   DATA[2032,33] := 0.3084905;
   DATA[2032,34] := 2.0;
   DATA[2032,35] := 250.2243;
   DATA[2032,36] := 1.69801;
   DATA[2032,37] := 189.1022;
   DATA[2032,38] := 0.000128152;
   DATA[2032,39] := 1.0;
   DATA[2032,40] := 1.0;
   DATA[2033,0] := 2.493034;
   DATA[2033,1] := 862.4616;
   DATA[2033,2] := 2.0;
   DATA[2033,3] := 2.0;
   DATA[2033,4] := 262.3686;
   DATA[2033,5] := 8.395155;
   DATA[2033,6] := 331.1971;
   DATA[2033,7] := 2.462179;
   DATA[2033,8] := 2.0;
   DATA[2033,9] := 2.0;
   DATA[2033,10] := 2.0;
   DATA[2033,11] := 19.76759;
   DATA[2033,12] := 2.209653;
   DATA[2033,13] := 801.3971;
   DATA[2033,14] := 1.0;
   DATA[2033,15] := 2.0;
   DATA[2033,16] := 1.0;
   DATA[2033,17] := 1.0;
   DATA[2033,18] := 1.0;
   DATA[2033,19] := 2.0;
   DATA[2033,20] := 148.808;
   DATA[2033,21] := 154.8834;
   DATA[2033,22] := 1.717361;
   DATA[2033,23] := 830.7485;
   DATA[2033,24] := 2.0;
   DATA[2033,25] := 2.0;
   DATA[2033,26] := 7.874455;
   DATA[2033,27] := 143.9375;
   DATA[2033,28] := 262.1764;
   DATA[2033,29] := 12.07383;
   DATA[2033,30] := 1.726609;
   DATA[2033,31] := 1.281798;
   DATA[2033,32] := 0.7355248;
   DATA[2033,33] := 0.3084905;
   DATA[2033,34] := 2.0;
   DATA[2033,35] := 250.2243;
   DATA[2033,36] := 1.69801;
   DATA[2033,37] := 189.0381;
   DATA[2033,38] := 0.000128152;
   DATA[2033,39] := 1.0;
   DATA[2033,40] := 1.0;
   DATA[2034,0] := 2.47702;
   DATA[2034,1] := 862.2653;
   DATA[2034,2] := 2.0;
   DATA[2034,3] := 2.0;
   DATA[2034,4] := 262.3686;
   DATA[2034,5] := 8.395155;
   DATA[2034,6] := 331.1971;
   DATA[2034,7] := 2.46282;
   DATA[2034,8] := 2.0;
   DATA[2034,9] := 2.0;
   DATA[2034,10] := 2.0;
   DATA[2034,11] := 19.74198;
   DATA[2034,12] := 2.208756;
   DATA[2034,13] := 801.6775;
   DATA[2034,14] := 1.0;
   DATA[2034,15] := 2.0;
   DATA[2034,16] := 1.0;
   DATA[2034,17] := 1.0;
   DATA[2034,18] := 1.0;
   DATA[2034,19] := 2.0;
   DATA[2034,20] := 148.808;
   DATA[2034,21] := 154.6783;
   DATA[2034,22] := 1.717361;
   DATA[2034,23] := 830.5947;
   DATA[2034,24] := 2.0;
   DATA[2034,25] := 2.0;
   DATA[2034,26] := 7.874455;
   DATA[2034,27] := 143.9375;
   DATA[2034,28] := 261.888;
   DATA[2034,29] := 12.07383;
   DATA[2034,30] := 1.725327;
   DATA[2034,31] := 1.277699;
   DATA[2034,32] := 0.7355248;
   DATA[2034,33] := 0.3084905;
   DATA[2034,34] := 2.0;
   DATA[2034,35] := 250.0641;
   DATA[2034,36] := 1.69801;
   DATA[2034,37] := 188.8779;
   DATA[2034,38] := 0.000128152;
   DATA[2034,39] := 1.0;
   DATA[2034,40] := 1.0;
   DATA[2035,0] := 2.456202;
   DATA[2035,1] := 862.1083;
   DATA[2035,2] := 2.0;
   DATA[2035,3] := 2.0;
   DATA[2035,4] := 262.3686;
   DATA[2035,5] := 8.395155;
   DATA[2035,6] := 331.1971;
   DATA[2035,7] := 2.46282;
   DATA[2035,8] := 2.0;
   DATA[2035,9] := 2.0;
   DATA[2035,10] := 2.0;
   DATA[2035,11] := 19.70997;
   DATA[2035,12] := 2.208756;
   DATA[2035,13] := 801.317;
   DATA[2035,14] := 1.0;
   DATA[2035,15] := 2.0;
   DATA[2035,16] := 1.0;
   DATA[2035,17] := 1.0;
   DATA[2035,18] := 1.0;
   DATA[2035,19] := 2.0;
   DATA[2035,20] := 148.808;
   DATA[2035,21] := 154.6783;
   DATA[2035,22] := 1.717361;
   DATA[2035,23] := 830.5563;
   DATA[2035,24] := 2.0;
   DATA[2035,25] := 2.0;
   DATA[2035,26] := 7.874455;
   DATA[2035,27] := 143.9375;
   DATA[2035,28] := 261.888;
   DATA[2035,29] := 12.07383;
   DATA[2035,30] := 1.723532;
   DATA[2035,31] := 1.260535;
   DATA[2035,32] := 0.7355248;
   DATA[2035,33] := 0.3084905;
   DATA[2035,34] := 2.0;
   DATA[2035,35] := 249.8558;
   DATA[2035,36] := 1.69801;
   DATA[2035,37] := 188.8138;
   DATA[2035,38] := 0.000128152;
   DATA[2035,39] := 1.0;
   DATA[2035,40] := 1.0;
   DATA[2036,0] := 2.445953;
   DATA[2036,1] := 862.2653;
   DATA[2036,2] := 2.0;
   DATA[2036,3] := 2.0;
   DATA[2036,4] := 262.3686;
   DATA[2036,5] := 8.395155;
   DATA[2036,6] := 331.1971;
   DATA[2036,7] := 2.463204;
   DATA[2036,8] := 2.0;
   DATA[2036,9] := 2.0;
   DATA[2036,10] := 2.0;
   DATA[2036,11] := 19.70997;
   DATA[2036,12] := 2.208756;
   DATA[2036,13] := 801.0767;
   DATA[2036,14] := 1.0;
   DATA[2036,15] := 2.0;
   DATA[2036,16] := 1.0;
   DATA[2036,17] := 1.0;
   DATA[2036,18] := 1.0;
   DATA[2036,19] := 2.0;
   DATA[2036,20] := 148.808;
   DATA[2036,21] := 154.6783;
   DATA[2036,22] := 1.716464;
   DATA[2036,23] := 831.1331;
   DATA[2036,24] := 2.0;
   DATA[2036,25] := 2.0;
   DATA[2036,26] := 7.874455;
   DATA[2036,27] := 143.9375;
   DATA[2036,28] := 261.888;
   DATA[2036,29] := 12.07383;
   DATA[2036,30] := 1.723532;
   DATA[2036,31] := 1.254259;
   DATA[2036,32] := 0.7355248;
   DATA[2036,33] := 0.3084905;
   DATA[2036,34] := 2.0;
   DATA[2036,35] := 249.8558;
   DATA[2036,36] := 1.69801;
   DATA[2036,37] := 188.8138;
   DATA[2036,38] := 0.000128152;
   DATA[2036,39] := 1.0;
   DATA[2036,40] := 1.0;
   DATA[2037,0] := 2.432822;
   DATA[2037,1] := 862.0691;
   DATA[2037,2] := 2.0;
   DATA[2037,3] := 2.0;
   DATA[2037,4] := 262.3686;
   DATA[2037,5] := 8.395155;
   DATA[2037,6] := 331.1971;
   DATA[2037,7] := 2.463589;
   DATA[2037,8] := 2.0;
   DATA[2037,9] := 2.0;
   DATA[2037,10] := 2.0;
   DATA[2037,11] := 19.75159;
   DATA[2037,12] := 2.208756;
   DATA[2037,13] := 801.1167;
   DATA[2037,14] := 1.0;
   DATA[2037,15] := 2.0;
   DATA[2037,16] := 1.0;
   DATA[2037,17] := 1.0;
   DATA[2037,18] := 1.0;
   DATA[2037,19] := 2.0;
   DATA[2037,20] := 148.808;
   DATA[2037,21] := 154.6783;
   DATA[2037,22] := 1.715824;
   DATA[2037,23] := 831.3253;
   DATA[2037,24] := 2.0;
   DATA[2037,25] := 2.0;
   DATA[2037,26] := 7.874455;
   DATA[2037,27] := 143.9375;
   DATA[2037,28] := 261.888;
   DATA[2037,29] := 12.07383;
   DATA[2037,30] := 1.723532;
   DATA[2037,31] := 1.241962;
   DATA[2037,32] := 0.7355248;
   DATA[2037,33] := 0.3077219;
   DATA[2037,34] := 2.0;
   DATA[2037,35] := 249.8558;
   DATA[2037,36] := 1.649953;
   DATA[2037,37] := 188.8138;
   DATA[2037,38] := 0.000128152;
   DATA[2037,39] := 1.0;
   DATA[2037,40] := 1.0;
   DATA[2038,0] := 2.432822;
   DATA[2038,1] := 862.0691;
   DATA[2038,2] := 2.0;
   DATA[2038,3] := 2.0;
   DATA[2038,4] := 262.3686;
   DATA[2038,5] := 8.395155;
   DATA[2038,6] := 331.1971;
   DATA[2038,7] := 2.463589;
   DATA[2038,8] := 2.0;
   DATA[2038,9] := 2.0;
   DATA[2038,10] := 2.0;
   DATA[2038,11] := 19.75159;
   DATA[2038,12] := 2.208756;
   DATA[2038,13] := 801.1167;
   DATA[2038,14] := 1.0;
   DATA[2038,15] := 2.0;
   DATA[2038,16] := 1.0;
   DATA[2038,17] := 1.0;
   DATA[2038,18] := 1.0;
   DATA[2038,19] := 2.0;
   DATA[2038,20] := 148.808;
   DATA[2038,21] := 154.6783;
   DATA[2038,22] := 1.715824;
   DATA[2038,23] := 831.3253;
   DATA[2038,24] := 2.0;
   DATA[2038,25] := 2.0;
   DATA[2038,26] := 7.874455;
   DATA[2038,27] := 143.9375;
   DATA[2038,28] := 261.888;
   DATA[2038,29] := 12.07383;
   DATA[2038,30] := 1.723532;
   DATA[2038,31] := 1.241962;
   DATA[2038,32] := 0.7355248;
   DATA[2038,33] := 0.3077219;
   DATA[2038,34] := 2.0;
   DATA[2038,35] := 249.8558;
   DATA[2038,36] := 1.649953;
   DATA[2038,37] := 188.8138;
   DATA[2038,38] := 0.000128152;
   DATA[2038,39] := 1.0;
   DATA[2038,40] := 1.0;
   DATA[2039,0] := 2.423213;
   DATA[2039,1] := 861.7158;
   DATA[2039,2] := 2.0;
   DATA[2039,3] := 2.0;
   DATA[2039,4] := 262.3686;
   DATA[2039,5] := 8.393232;
   DATA[2039,6] := 331.1971;
   DATA[2039,7] := 2.463589;
   DATA[2039,8] := 2.0;
   DATA[2039,9] := 2.0;
   DATA[2039,10] := 2.0;
   DATA[2039,11] := 19.77399;
   DATA[2039,12] := 2.210037;
   DATA[2039,13] := 800.9565;
   DATA[2039,14] := 1.0;
   DATA[2039,15] := 2.0;
   DATA[2039,16] := 1.0;
   DATA[2039,17] := 1.0;
   DATA[2039,18] := 1.0;
   DATA[2039,19] := 2.0;
   DATA[2039,20] := 148.808;
   DATA[2039,21] := 154.909;
   DATA[2039,22] := 1.715824;
   DATA[2039,23] := 831.3253;
   DATA[2039,24] := 2.0;
   DATA[2039,25] := 2.0;
   DATA[2039,26] := 7.874455;
   DATA[2039,27] := 143.9375;
   DATA[2039,28] := 261.888;
   DATA[2039,29] := 12.07383;
   DATA[2039,30] := 1.725455;
   DATA[2039,31] := 1.237351;
   DATA[2039,32] := 0.7355248;
   DATA[2039,33] := 0.3077219;
   DATA[2039,34] := 2.0;
   DATA[2039,35] := 250.032;
   DATA[2039,36] := 1.649953;
   DATA[2039,37] := 188.8138;
   DATA[2039,38] := 0.000128152;
   DATA[2039,39] := 1.0;
   DATA[2039,40] := 1.0;
   DATA[2040,0] := 2.423213;
   DATA[2040,1] := 862.0691;
   DATA[2040,2] := 2.0;
   DATA[2040,3] := 2.0;
   DATA[2040,4] := 262.3686;
   DATA[2040,5] := 8.393232;
   DATA[2040,6] := 331.1971;
   DATA[2040,7] := 2.463589;
   DATA[2040,8] := 2.0;
   DATA[2040,9] := 2.0;
   DATA[2040,10] := 2.0;
   DATA[2040,11] := 19.77399;
   DATA[2040,12] := 2.210037;
   DATA[2040,13] := 800.7562;
   DATA[2040,14] := 1.0;
   DATA[2040,15] := 2.0;
   DATA[2040,16] := 1.0;
   DATA[2040,17] := 1.0;
   DATA[2040,18] := 1.0;
   DATA[2040,19] := 2.0;
   DATA[2040,20] := 148.808;
   DATA[2040,21] := 155.0372;
   DATA[2040,22] := 1.715824;
   DATA[2040,23] := 831.556;
   DATA[2040,24] := 2.0;
   DATA[2040,25] := 2.0;
   DATA[2040,26] := 7.874455;
   DATA[2040,27] := 143.9375;
   DATA[2040,28] := 262.1764;
   DATA[2040,29] := 12.07383;
   DATA[2040,30] := 1.725583;
   DATA[2040,31] := 1.251953;
   DATA[2040,32] := 0.7355248;
   DATA[2040,33] := 0.3084905;
   DATA[2040,34] := 2.0;
   DATA[2040,35] := 250.0961;
   DATA[2040,36] := 1.649953;
   DATA[2040,37] := 188.9419;
   DATA[2040,38] := 0.000128152;
   DATA[2040,39] := 1.0;
   DATA[2040,40] := 1.0;
   DATA[2041,0] := 2.433783;
   DATA[2041,1] := 861.598;
   DATA[2041,2] := 2.0;
   DATA[2041,3] := 2.0;
   DATA[2041,4] := 262.3686;
   DATA[2041,5] := 8.393232;
   DATA[2041,6] := 331.0946;
   DATA[2041,7] := 2.463589;
   DATA[2041,8] := 2.0;
   DATA[2041,9] := 2.0;
   DATA[2041,10] := 2.0;
   DATA[2041,11] := 19.77399;
   DATA[2041,12] := 2.210037;
   DATA[2041,13] := 800.7162;
   DATA[2041,14] := 1.0;
   DATA[2041,15] := 2.0;
   DATA[2041,16] := 1.0;
   DATA[2041,17] := 1.0;
   DATA[2041,18] := 1.0;
   DATA[2041,19] := 2.0;
   DATA[2041,20] := 148.808;
   DATA[2041,21] := 155.0372;
   DATA[2041,22] := 1.718387;
   DATA[2041,23] := 831.5176;
   DATA[2041,24] := 2.0;
   DATA[2041,25] := 2.0;
   DATA[2041,26] := 7.874455;
   DATA[2041,27] := 143.9375;
   DATA[2041,28] := 262.1764;
   DATA[2041,29] := 12.07383;
   DATA[2041,30] := 1.726096;
   DATA[2041,31] := 1.267837;
   DATA[2041,32] := 0.7355248;
   DATA[2041,33] := 0.3084905;
   DATA[2041,34] := 2.0;
   DATA[2041,35] := 250.1923;
   DATA[2041,36] := 1.649953;
   DATA[2041,37] := 189.1342;
   DATA[2041,38] := 0.000128152;
   DATA[2041,39] := 1.0;
   DATA[2041,40] := 1.0;
   DATA[2042,0] := 2.487589;
   DATA[2042,1] := 861.6373;
   DATA[2042,2] := 2.0;
   DATA[2042,3] := 2.0;
   DATA[2042,4] := 262.3686;
   DATA[2042,5] := 8.393232;
   DATA[2042,6] := 331.0946;
   DATA[2042,7] := 2.463589;
   DATA[2042,8] := 2.0;
   DATA[2042,9] := 2.0;
   DATA[2042,10] := 2.0;
   DATA[2042,11] := 19.74198;
   DATA[2042,12] := 2.210037;
   DATA[2042,13] := 800.5159;
   DATA[2042,14] := 1.0;
   DATA[2042,15] := 2.0;
   DATA[2042,16] := 1.0;
   DATA[2042,17] := 1.0;
   DATA[2042,18] := 1.0;
   DATA[2042,19] := 2.0;
   DATA[2042,20] := 148.808;
   DATA[2042,21] := 154.8065;
   DATA[2042,22] := 1.718387;
   DATA[2042,23] := 831.7098;
   DATA[2042,24] := 2.0;
   DATA[2042,25] := 2.0;
   DATA[2042,26] := 7.874455;
   DATA[2042,27] := 143.9375;
   DATA[2042,28] := 262.1764;
   DATA[2042,29] := 12.07383;
   DATA[2042,30] := 1.728275;
   DATA[2042,31] := 1.280646;
   DATA[2042,32] := 0.7355248;
   DATA[2042,33] := 0.3070813;
   DATA[2042,34] := 2.0;
   DATA[2042,35] := 250.4005;
   DATA[2042,36] := 1.649953;
   DATA[2042,37] := 189.1662;
   DATA[2042,38] := 0.000128152;
   DATA[2042,39] := 1.0;
   DATA[2042,40] := 1.0;
   DATA[2043,0] := 2.531147;
   DATA[2043,1] := 861.3232;
   DATA[2043,2] := 2.0;
   DATA[2043,3] := 2.0;
   DATA[2043,4] := 262.3686;
   DATA[2043,5] := 8.393232;
   DATA[2043,6] := 331.0946;
   DATA[2043,7] := 2.461667;
   DATA[2043,8] := 2.0;
   DATA[2043,9] := 2.0;
   DATA[2043,10] := 2.0;
   DATA[2043,11] := 19.72598;
   DATA[2043,12] := 2.210037;
   DATA[2043,13] := 800.7162;
   DATA[2043,14] := 1.0;
   DATA[2043,15] := 2.0;
   DATA[2043,16] := 1.0;
   DATA[2043,17] := 1.0;
   DATA[2043,18] := 1.0;
   DATA[2043,19] := 2.0;
   DATA[2043,20] := 148.808;
   DATA[2043,21] := 154.8065;
   DATA[2043,22] := 1.718387;
   DATA[2043,23] := 831.556;
   DATA[2043,24] := 2.0;
   DATA[2043,25] := 2.0;
   DATA[2043,26] := 7.874455;
   DATA[2043,27] := 143.9375;
   DATA[2043,28] := 262.0802;
   DATA[2043,29] := 12.07383;
   DATA[2043,30] := 1.728275;
   DATA[2043,31] := 1.281798;
   DATA[2043,32] := 0.7355248;
   DATA[2043,33] := 0.3068251;
   DATA[2043,34] := 2.0;
   DATA[2043,35] := 250.4005;
   DATA[2043,36] := 1.649953;
   DATA[2043,37] := 189.1662;
   DATA[2043,38] := 0.000128152;
   DATA[2043,39] := 1.0;
   DATA[2043,40] := 1.0;
   DATA[2044,0] := 2.573744;
   DATA[2044,1] := 861.5195;
   DATA[2044,2] := 2.0;
   DATA[2044,3] := 2.0;
   DATA[2044,4] := 262.3686;
   DATA[2044,5] := 8.393232;
   DATA[2044,6] := 331.0946;
   DATA[2044,7] := 2.461667;
   DATA[2044,8] := 2.0;
   DATA[2044,9] := 2.0;
   DATA[2044,10] := 2.0;
   DATA[2044,11] := 19.72598;
   DATA[2044,12] := 2.210037;
   DATA[2044,13] := 800.5159;
   DATA[2044,14] := 1.0;
   DATA[2044,15] := 2.0;
   DATA[2044,16] := 1.0;
   DATA[2044,17] := 1.0;
   DATA[2044,18] := 1.0;
   DATA[2044,19] := 2.0;
   DATA[2044,20] := 148.808;
   DATA[2044,21] := 154.8065;
   DATA[2044,22] := 1.718387;
   DATA[2044,23] := 831.6329;
   DATA[2044,24] := 2.0;
   DATA[2044,25] := 2.0;
   DATA[2044,26] := 7.874455;
   DATA[2044,27] := 143.9375;
   DATA[2044,28] := 262.0802;
   DATA[2044,29] := 12.07383;
   DATA[2044,30] := 1.730069;
   DATA[2044,31] := 1.271935;
   DATA[2044,32] := 0.7355248;
   DATA[2044,33] := 0.3068251;
   DATA[2044,34] := 2.0;
   DATA[2044,35] := 250.4005;
   DATA[2044,36] := 1.746067;
   DATA[2044,37] := 189.2624;
   DATA[2044,38] := 0.000128152;
   DATA[2044,39] := 1.0;
   DATA[2044,40] := 1.0;
   DATA[2045,0] := 2.601928;
   DATA[2045,1] := 861.5195;
   DATA[2045,2] := 2.0;
   DATA[2045,3] := 2.0;
   DATA[2045,4] := 262.3686;
   DATA[2045,5] := 8.393232;
   DATA[2045,6] := 331.0946;
   DATA[2045,7] := 2.461667;
   DATA[2045,8] := 2.0;
   DATA[2045,9] := 2.0;
   DATA[2045,10] := 2.0;
   DATA[2045,11] := 19.72598;
   DATA[2045,12] := 2.210037;
   DATA[2045,13] := 800.3156;
   DATA[2045,14] := 1.0;
   DATA[2045,15] := 2.0;
   DATA[2045,16] := 1.0;
   DATA[2045,17] := 1.0;
   DATA[2045,18] := 1.0;
   DATA[2045,19] := 2.0;
   DATA[2045,20] := 148.808;
   DATA[2045,21] := 154.8065;
   DATA[2045,22] := 1.718387;
   DATA[2045,23] := 831.7867;
   DATA[2045,24] := 2.0;
   DATA[2045,25] := 2.0;
   DATA[2045,26] := 7.874455;
   DATA[2045,27] := 144.2451;
   DATA[2045,28] := 262.0802;
   DATA[2045,29] := 12.07383;
   DATA[2045,30] := 1.731351;
   DATA[2045,31] := 1.271935;
   DATA[2045,32] := 0.7355248;
   DATA[2045,33] := 0.3068251;
   DATA[2045,34] := 2.0;
   DATA[2045,35] := 250.5127;
   DATA[2045,36] := 1.762086;
   DATA[2045,37] := 189.2624;
   DATA[2045,38] := 0.000128152;
   DATA[2045,39] := 1.0;
   DATA[2045,40] := 1.0;
   DATA[2046,0] := 2.636198;
   DATA[2046,1] := 861.284;
   DATA[2046,2] := 2.0;
   DATA[2046,3] := 2.0;
   DATA[2046,4] := 262.3686;
   DATA[2046,5] := 8.393232;
   DATA[2046,6] := 331.0946;
   DATA[2046,7] := 2.461667;
   DATA[2046,8] := 2.0;
   DATA[2046,9] := 2.0;
   DATA[2046,10] := 2.0;
   DATA[2046,11] := 19.71957;
   DATA[2046,12] := 2.206963;
   DATA[2046,13] := 800.3958;
   DATA[2046,14] := 1.0;
   DATA[2046,15] := 2.0;
   DATA[2046,16] := 1.0;
   DATA[2046,17] := 1.0;
   DATA[2046,18] := 1.0;
   DATA[2046,19] := 2.0;
   DATA[2046,20] := 148.808;
   DATA[2046,21] := 154.8065;
   DATA[2046,22] := 1.718387;
   DATA[2046,23] := 832.3635;
   DATA[2046,24] := 2.0;
   DATA[2046,25] := 2.0;
   DATA[2046,26] := 7.874455;
   DATA[2046,27] := 144.2451;
   DATA[2046,28] := 262.0802;
   DATA[2046,29] := 12.07383;
   DATA[2046,30] := 1.731351;
   DATA[2046,31] := 1.271679;
   DATA[2046,32] := 0.7355248;
   DATA[2046,33] := 0.3068251;
   DATA[2046,34] := 2.0;
   DATA[2046,35] := 250.6409;
   DATA[2046,36] := 1.762086;
   DATA[2046,37] := 189.3585;
   DATA[2046,38] := 0.000128152;
   DATA[2046,39] := 1.0;
   DATA[2046,40] := 1.0;
   DATA[2047,0] := 2.653172;
   DATA[2047,1] := 861.441;
   DATA[2047,2] := 2.0;
   DATA[2047,3] := 2.0;
   DATA[2047,4] := 262.3686;
   DATA[2047,5] := 8.393232;
   DATA[2047,6] := 331.0946;
   DATA[2047,7] := 2.461667;
   DATA[2047,8] := 2.0;
   DATA[2047,9] := 2.0;
   DATA[2047,10] := 2.0;
   DATA[2047,11] := 19.71957;
   DATA[2047,12] := 2.206322;
   DATA[2047,13] := 800.3156;
   DATA[2047,14] := 1.0;
   DATA[2047,15] := 2.0;
   DATA[2047,16] := 1.0;
   DATA[2047,17] := 1.0;
   DATA[2047,18] := 1.0;
   DATA[2047,19] := 2.0;
   DATA[2047,20] := 148.808;
   DATA[2047,21] := 154.8065;
   DATA[2047,22] := 1.718387;
   DATA[2047,23] := 832.2866;
   DATA[2047,24] := 2.0;
   DATA[2047,25] := 2.0;
   DATA[2047,26] := 7.874455;
   DATA[2047,27] := 144.0913;
   DATA[2047,28] := 262.0802;
   DATA[2047,29] := 12.07383;
   DATA[2047,30] := 1.731351;
   DATA[2047,31] := 1.290637;
   DATA[2047,32] := 0.7355248;
   DATA[2047,33] := 0.3068251;
   DATA[2047,34] := 2.0;
   DATA[2047,35] := 250.6409;
   DATA[2047,36] := 1.681991;
   DATA[2047,37] := 189.4386;
   DATA[2047,38] := 0.000128152;
   DATA[2047,39] := 1.0;
   DATA[2047,40] := 1.0;
   DATA[2048,0] := 2.663421;
   DATA[2048,1] := 861.441;
   DATA[2048,2] := 2.0;
   DATA[2048,3] := 2.0;
   DATA[2048,4] := 262.3686;
   DATA[2048,5] := 8.393232;
   DATA[2048,6] := 331.0946;
   DATA[2048,7] := 2.461667;
   DATA[2048,8] := 2.0;
   DATA[2048,9] := 2.0;
   DATA[2048,10] := 2.0;
   DATA[2048,11] := 19.69396;
   DATA[2048,12] := 2.206322;
   DATA[2048,13] := 800.3156;
   DATA[2048,14] := 1.0;
   DATA[2048,15] := 2.0;
   DATA[2048,16] := 1.0;
   DATA[2048,17] := 1.0;
   DATA[2048,18] := 1.0;
   DATA[2048,19] := 2.0;
   DATA[2048,20] := 148.808;
   DATA[2048,21] := 155.0372;
   DATA[2048,22] := 1.718387;
   DATA[2048,23] := 832.3635;
   DATA[2048,24] := 2.0;
   DATA[2048,25] := 2.0;
   DATA[2048,26] := 7.874455;
   DATA[2048,27] := 143.8862;
   DATA[2048,28] := 262.0802;
   DATA[2048,29] := 12.07383;
   DATA[2048,30] := 1.731351;
   DATA[2048,31] := 1.291789;
   DATA[2048,32] := 0.7355248;
   DATA[2048,33] := 0.3063127;
   DATA[2048,34] := 2.0;
   DATA[2048,35] := 250.6248;
   DATA[2048,36] := 1.649953;
   DATA[2048,37] := 189.4386;
   DATA[2048,38] := 0.000128152;
   DATA[2048,39] := 1.0;
   DATA[2048,40] := 1.0;
   DATA[2049,0] := 2.664062;
   DATA[2049,1] := 861.284;
   DATA[2049,2] := 2.0;
   DATA[2049,3] := 2.0;
   DATA[2049,4] := 262.3686;
   DATA[2049,5] := 8.393232;
   DATA[2049,6] := 331.0946;
   DATA[2049,7] := 2.461667;
   DATA[2049,8] := 2.0;
   DATA[2049,9] := 2.0;
   DATA[2049,10] := 2.0;
   DATA[2049,11] := 19.67796;
   DATA[2049,12] := 2.206322;
   DATA[2049,13] := 800.596;
   DATA[2049,14] := 1.0;
   DATA[2049,15] := 2.0;
   DATA[2049,16] := 1.0;
   DATA[2049,17] := 1.0;
   DATA[2049,18] := 1.0;
   DATA[2049,19] := 2.0;
   DATA[2049,20] := 148.808;
   DATA[2049,21] := 155.0372;
   DATA[2049,22] := 1.715952;
   DATA[2049,23] := 832.9018;
   DATA[2049,24] := 2.0;
   DATA[2049,25] := 2.0;
   DATA[2049,26] := 7.874455;
   DATA[2049,27] := 143.8862;
   DATA[2049,28] := 262.0802;
   DATA[2049,29] := 12.07383;
   DATA[2049,30] := 1.730838;
   DATA[2049,31] := 1.291918;
   DATA[2049,32] := 0.7355248;
   DATA[2049,33] := 0.3063127;
   DATA[2049,34] := 2.0;
   DATA[2049,35] := 250.3525;
   DATA[2049,36] := 1.649953;
   DATA[2049,37] := 189.3265;
   DATA[2049,38] := 0.000128152;
   DATA[2049,39] := 1.0;
   DATA[2049,40] := 1.0;
   DATA[2050,0] := 2.628191;
   DATA[2050,1] := 861.6373;
   DATA[2050,2] := 2.0;
   DATA[2050,3] := 2.0;
   DATA[2050,4] := 262.3686;
   DATA[2050,5] := 8.393232;
   DATA[2050,6] := 331.0946;
   DATA[2050,7] := 2.463589;
   DATA[2050,8] := 2.0;
   DATA[2050,9] := 2.0;
   DATA[2050,10] := 2.0;
   DATA[2050,11] := 19.67796;
   DATA[2050,12] := 2.206322;
   DATA[2050,13] := 800.7162;
   DATA[2050,14] := 1.0;
   DATA[2050,15] := 2.0;
   DATA[2050,16] := 1.0;
   DATA[2050,17] := 1.0;
   DATA[2050,18] := 1.0;
   DATA[2050,19] := 2.0;
   DATA[2050,20] := 148.808;
   DATA[2050,21] := 155.0372;
   DATA[2050,22] := 1.715952;
   DATA[2050,23] := 832.7095;
   DATA[2050,24] := 2.0;
   DATA[2050,25] := 2.0;
   DATA[2050,26] := 7.874455;
   DATA[2050,27] := 143.8862;
   DATA[2050,28] := 262.0802;
   DATA[2050,29] := 12.07383;
   DATA[2050,30] := 1.728019;
   DATA[2050,31] := 1.286922;
   DATA[2050,32] := 0.7355248;
   DATA[2050,33] := 0.3063127;
   DATA[2050,34] := 2.0;
   DATA[2050,35] := 250.3525;
   DATA[2050,36] := 1.649953;
   DATA[2050,37] := 189.1823;
   DATA[2050,38] := 0.000128152;
   DATA[2050,39] := 1.0;
   DATA[2050,40] := 1.0;
   DATA[2051,0] := 2.620824;
   DATA[2051,1] := 861.441;
   DATA[2051,2] := 2.0;
   DATA[2051,3] := 2.0;
   DATA[2051,4] := 262.3686;
   DATA[2051,5] := 8.392271;
   DATA[2051,6] := 331.0946;
   DATA[2051,7] := 2.463589;
   DATA[2051,8] := 2.0;
   DATA[2051,9] := 2.0;
   DATA[2051,10] := 2.0;
   DATA[2051,11] := 19.67796;
   DATA[2051,12] := 2.206322;
   DATA[2051,13] := 800.7963;
   DATA[2051,14] := 1.0;
   DATA[2051,15] := 2.0;
   DATA[2051,16] := 1.0;
   DATA[2051,17] := 1.0;
   DATA[2051,18] := 1.0;
   DATA[2051,19] := 2.0;
   DATA[2051,20] := 148.808;
   DATA[2051,21] := 155.0372;
   DATA[2051,22] := 1.715952;
   DATA[2051,23] := 833.171;
   DATA[2051,24] := 2.0;
   DATA[2051,25] := 2.0;
   DATA[2051,26] := 7.874455;
   DATA[2051,27] := 143.8862;
   DATA[2051,28] := 262.0802;
   DATA[2051,29] := 12.07383;
   DATA[2051,30] := 1.726865;
   DATA[2051,31] := 1.280902;
   DATA[2051,32] := 0.7355248;
   DATA[2051,33] := 0.3063127;
   DATA[2051,34] := 2.0;
   DATA[2051,35] := 250.3525;
   DATA[2051,36] := 1.649953;
   DATA[2051,37] := 189.1022;
   DATA[2051,38] := 0.000128152;
   DATA[2051,39] := 1.0;
   DATA[2051,40] := 1.0;
   DATA[2052,0] := 2.61538;
   DATA[2052,1] := 861.6765;
   DATA[2052,2] := 2.0;
   DATA[2052,3] := 2.0;
   DATA[2052,4] := 262.3686;
   DATA[2052,5] := 8.392271;
   DATA[2052,6] := 331.0946;
   DATA[2052,7] := 2.465127;
   DATA[2052,8] := 2.0;
   DATA[2052,9] := 2.0;
   DATA[2052,10] := 2.0;
   DATA[2052,11] := 19.62674;
   DATA[2052,12] := 2.206707;
   DATA[2052,13] := 801.1167;
   DATA[2052,14] := 1.0;
   DATA[2052,15] := 2.0;
   DATA[2052,16] := 1.0;
   DATA[2052,17] := 1.0;
   DATA[2052,18] := 1.0;
   DATA[2052,19] := 2.0;
   DATA[2052,20] := 148.808;
   DATA[2052,21] := 155.0372;
   DATA[2052,22] := 1.715952;
   DATA[2052,23] := 832.9787;
   DATA[2052,24] := 2.0;
   DATA[2052,25] := 2.0;
   DATA[2052,26] := 7.874455;
   DATA[2052,27] := 143.9631;
   DATA[2052,28] := 262.0802;
   DATA[2052,29] := 12.07383;
   DATA[2052,30] := 1.726609;
   DATA[2052,31] := 1.280902;
   DATA[2052,32] := 0.7355248;
   DATA[2052,33] := 0.3084265;
   DATA[2052,34] := 2.0;
   DATA[2052,35] := 250.3044;
   DATA[2052,36] := 1.649953;
   DATA[2052,37] := 189.1022;
   DATA[2052,38] := 0.000128152;
   DATA[2052,39] := 1.0;
   DATA[2052,40] := 1.0;
   DATA[2053,0] := 2.606732;
   DATA[2053,1] := 861.284;
   DATA[2053,2] := 2.0;
   DATA[2053,3] := 2.0;
   DATA[2053,4] := 262.3686;
   DATA[2053,5] := 8.392271;
   DATA[2053,6] := 331.0946;
   DATA[2053,7] := 2.465127;
   DATA[2053,8] := 2.0;
   DATA[2053,9] := 2.0;
   DATA[2053,10] := 2.0;
   DATA[2053,11] := 19.62674;
   DATA[2053,12] := 2.207091;
   DATA[2053,13] := 800.7963;
   DATA[2053,14] := 1.0;
   DATA[2053,15] := 2.0;
   DATA[2053,16] := 1.0;
   DATA[2053,17] := 1.0;
   DATA[2053,18] := 1.0;
   DATA[2053,19] := 2.0;
   DATA[2053,20] := 148.808;
   DATA[2053,21] := 155.0372;
   DATA[2053,22] := 1.716592;
   DATA[2053,23] := 833.1325;
   DATA[2053,24] := 2.0;
   DATA[2053,25] := 2.0;
   DATA[2053,26] := 7.874455;
   DATA[2053,27] := 143.9631;
   DATA[2053,28] := 262.0802;
   DATA[2053,29] := 12.07383;
   DATA[2053,30] := 1.726609;
   DATA[2053,31] := 1.274881;
   DATA[2053,32] := 0.7355248;
   DATA[2053,33] := 0.3084265;
   DATA[2053,34] := 2.0;
   DATA[2053,35] := 250.3044;
   DATA[2053,36] := 1.730048;
   DATA[2053,37] := 189.1022;
   DATA[2053,38] := 0.000128152;
   DATA[2053,39] := 1.0;
   DATA[2053,40] := 1.0;
   DATA[2054,0] := 2.582071;
   DATA[2054,1] := 861.5195;
   DATA[2054,2] := 2.0;
   DATA[2054,3] := 2.0;
   DATA[2054,4] := 262.3686;
   DATA[2054,5] := 8.392271;
   DATA[2054,6] := 331.0946;
   DATA[2054,7] := 2.464742;
   DATA[2054,8] := 2.0;
   DATA[2054,9] := 2.0;
   DATA[2054,10] := 2.0;
   DATA[2054,11] := 19.62674;
   DATA[2054,12] := 2.209013;
   DATA[2054,13] := 801.3971;
   DATA[2054,14] := 1.0;
   DATA[2054,15] := 2.0;
   DATA[2054,16] := 1.0;
   DATA[2054,17] := 1.0;
   DATA[2054,18] := 1.0;
   DATA[2054,19] := 2.0;
   DATA[2054,20] := 148.808;
   DATA[2054,21] := 155.0372;
   DATA[2054,22] := 1.717361;
   DATA[2054,23] := 832.9402;
   DATA[2054,24] := 2.0;
   DATA[2054,25] := 2.0;
   DATA[2054,26] := 7.874455;
   DATA[2054,27] := 143.9631;
   DATA[2054,28] := 262.0802;
   DATA[2054,29] := 12.07383;
   DATA[2054,30] := 1.726609;
   DATA[2054,31] := 1.276162;
   DATA[2054,32] := 0.7355248;
   DATA[2054,33] := 0.3084265;
   DATA[2054,34] := 2.0;
   DATA[2054,35] := 250.3044;
   DATA[2054,36] := 1.730048;
   DATA[2054,37] := 189.1022;
   DATA[2054,38] := 0.000128152;
   DATA[2054,39] := 1.0;
   DATA[2054,40] := 1.0;
   DATA[2055,0] := 2.564456;
   DATA[2055,1] := 861.284;
   DATA[2055,2] := 2.0;
   DATA[2055,3] := 2.0;
   DATA[2055,4] := 262.3686;
   DATA[2055,5] := 8.392271;
   DATA[2055,6] := 331.0946;
   DATA[2055,7] := 2.463589;
   DATA[2055,8] := 2.0;
   DATA[2055,9] := 2.0;
   DATA[2055,10] := 2.0;
   DATA[2055,11] := 19.69396;
   DATA[2055,12] := 2.209653;
   DATA[2055,13] := 801.5173;
   DATA[2055,14] := 1.0;
   DATA[2055,15] := 2.0;
   DATA[2055,16] := 1.0;
   DATA[2055,17] := 1.0;
   DATA[2055,18] := 1.0;
   DATA[2055,19] := 2.0;
   DATA[2055,20] := 148.808;
   DATA[2055,21] := 154.8321;
   DATA[2055,22] := 1.717746;
   DATA[2055,23] := 833.4786;
   DATA[2055,24] := 2.0;
   DATA[2055,25] := 2.0;
   DATA[2055,26] := 7.874455;
   DATA[2055,27] := 143.9631;
   DATA[2055,28] := 262.0802;
   DATA[2055,29] := 12.07383;
   DATA[2055,30] := 1.726609;
   DATA[2055,31] := 1.277315;
   DATA[2055,32] := 0.7355248;
   DATA[2055,33] := 0.3084265;
   DATA[2055,34] := 2.0;
   DATA[2055,35] := 250.3044;
   DATA[2055,36] := 1.730048;
   DATA[2055,37] := 189.1022;
   DATA[2055,38] := 0.000128152;
   DATA[2055,39] := 1.0;
   DATA[2055,40] := 1.0;
   DATA[2056,0] := 2.544919;
   DATA[2056,1] := 861.598;
   DATA[2056,2] := 2.0;
   DATA[2056,3] := 2.0;
   DATA[2056,4] := 262.3686;
   DATA[2056,5] := 8.392271;
   DATA[2056,6] := 331.0946;
   DATA[2056,7] := 2.463589;
   DATA[2056,8] := 2.0;
   DATA[2056,9] := 2.0;
   DATA[2056,10] := 2.0;
   DATA[2056,11] := 19.70357;
   DATA[2056,12] := 2.209653;
   DATA[2056,13] := 801.7576;
   DATA[2056,14] := 1.0;
   DATA[2056,15] := 2.0;
   DATA[2056,16] := 1.0;
   DATA[2056,17] := 1.0;
   DATA[2056,18] := 1.0;
   DATA[2056,19] := 2.0;
   DATA[2056,20] := 148.808;
   DATA[2056,21] := 154.8321;
   DATA[2056,22] := 1.717746;
   DATA[2056,23] := 833.3248;
   DATA[2056,24] := 2.0;
   DATA[2056,25] := 2.0;
   DATA[2056,26] := 7.874455;
   DATA[2056,27] := 143.9631;
   DATA[2056,28] := 262.0802;
   DATA[2056,29] := 12.07383;
   DATA[2056,30] := 1.726609;
   DATA[2056,31] := 1.269758;
   DATA[2056,32] := 0.7355248;
   DATA[2056,33] := 0.3084265;
   DATA[2056,34] := 2.0;
   DATA[2056,35] := 250.3044;
   DATA[2056,36] := 1.730048;
   DATA[2056,37] := 189.1983;
   DATA[2056,38] := 0.000128152;
   DATA[2056,39] := 1.0;
   DATA[2056,40] := 1.0;
   DATA[2057,0] := 2.529546;
   DATA[2057,1] := 861.2448;
   DATA[2057,2] := 2.0;
   DATA[2057,3] := 2.0;
   DATA[2057,4] := 262.3686;
   DATA[2057,5] := 8.392271;
   DATA[2057,6] := 331.0946;
   DATA[2057,7] := 2.461667;
   DATA[2057,8] := 2.0;
   DATA[2057,9] := 2.0;
   DATA[2057,10] := 2.0;
   DATA[2057,11] := 19.73238;
   DATA[2057,12] := 2.209653;
   DATA[2057,13] := 802.2783;
   DATA[2057,14] := 1.0;
   DATA[2057,15] := 2.0;
   DATA[2057,16] := 1.0;
   DATA[2057,17] := 1.0;
   DATA[2057,18] := 1.0;
   DATA[2057,19] := 2.0;
   DATA[2057,20] := 148.808;
   DATA[2057,21] := 154.8321;
   DATA[2057,22] := 1.718643;
   DATA[2057,23] := 833.94;
   DATA[2057,24] := 2.0;
   DATA[2057,25] := 2.0;
   DATA[2057,26] := 7.874455;
   DATA[2057,27] := 143.9631;
   DATA[2057,28] := 262.0802;
   DATA[2057,29] := 12.07383;
   DATA[2057,30] := 1.72725;
   DATA[2057,31] := 1.279877;
   DATA[2057,32] := 0.7351407;
   DATA[2057,33] := 0.3084265;
   DATA[2057,34] := 2.0;
   DATA[2057,35] := 250.4807;
   DATA[2057,36] := 1.730048;
   DATA[2057,37] := 189.4386;
   DATA[2057,38] := 0.000128152;
   DATA[2057,39] := 1.0;
   DATA[2057,40] := 1.0;
   DATA[2058,0] := 2.508407;
   DATA[2058,1] := 861.598;
   DATA[2058,2] := 2.0;
   DATA[2058,3] := 2.0;
   DATA[2058,4] := 262.3686;
   DATA[2058,5] := 8.392271;
   DATA[2058,6] := 331.0946;
   DATA[2058,7] := 2.461667;
   DATA[2058,8] := 2.0;
   DATA[2058,9] := 2.0;
   DATA[2058,10] := 2.0;
   DATA[2058,11] := 19.76439;
   DATA[2058,12] := 2.209653;
   DATA[2058,13] := 802.5186;
   DATA[2058,14] := 1.0;
   DATA[2058,15] := 2.0;
   DATA[2058,16] := 1.0;
   DATA[2058,17] := 1.0;
   DATA[2058,18] := 1.0;
   DATA[2058,19] := 2.0;
   DATA[2058,20] := 148.808;
   DATA[2058,21] := 154.8321;
   DATA[2058,22] := 1.719156;
   DATA[2058,23] := 834.0938;
   DATA[2058,24] := 2.0;
   DATA[2058,25] := 2.0;
   DATA[2058,26] := 7.874455;
   DATA[2058,27] := 143.9631;
   DATA[2058,28] := 262.0802;
   DATA[2058,29] := 12.07383;
   DATA[2058,30] := 1.728916;
   DATA[2058,31] := 1.28167;
   DATA[2058,32] := 0.7348846;
   DATA[2058,33] := 0.3084265;
   DATA[2058,34] := 2.0;
   DATA[2058,35] := 250.5928;
   DATA[2058,36] := 1.730048;
   DATA[2058,37] := 189.4386;
   DATA[2058,38] := 0.000128152;
   DATA[2058,39] := 1.0;
   DATA[2058,40] := 1.0;
   DATA[2059,0] := 2.496237;
   DATA[2059,1] := 861.441;
   DATA[2059,2] := 2.0;
   DATA[2059,3] := 2.0;
   DATA[2059,4] := 262.3686;
   DATA[2059,5] := 8.392271;
   DATA[2059,6] := 331.0946;
   DATA[2059,7] := 2.461667;
   DATA[2059,8] := 2.0;
   DATA[2059,9] := 2.0;
   DATA[2059,10] := 2.0;
   DATA[2059,11] := 19.76439;
   DATA[2059,12] := 2.209653;
   DATA[2059,13] := 802.4786;
   DATA[2059,14] := 1.0;
   DATA[2059,15] := 2.0;
   DATA[2059,16] := 1.0;
   DATA[2059,17] := 1.0;
   DATA[2059,18] := 1.0;
   DATA[2059,19] := 2.0;
   DATA[2059,20] := 148.808;
   DATA[2059,21] := 154.8321;
   DATA[2059,22] := 1.719156;
   DATA[2059,23] := 834.2092;
   DATA[2059,24] := 2.0;
   DATA[2059,25] := 2.0;
   DATA[2059,26] := 7.874455;
   DATA[2059,27] := 143.9631;
   DATA[2059,28] := 262.0161;
   DATA[2059,29] := 12.07383;
   DATA[2059,30] := 1.728916;
   DATA[2059,31] := 1.299219;
   DATA[2059,32] := 0.7348846;
   DATA[2059,33] := 0.3068891;
   DATA[2059,34] := 2.0;
   DATA[2059,35] := 250.5928;
   DATA[2059,36] := 1.730048;
   DATA[2059,37] := 189.4386;
   DATA[2059,38] := 0.000128152;
   DATA[2059,39] := 1.0;
   DATA[2059,40] := 1.0;
   DATA[2060,0] := 2.478301;
   DATA[2060,1] := 861.3232;
   DATA[2060,2] := 2.0;
   DATA[2060,3] := 2.0;
   DATA[2060,4] := 262.3686;
   DATA[2060,5] := 8.392271;
   DATA[2060,6] := 331.0946;
   DATA[2060,7] := 2.461667;
   DATA[2060,8] := 2.0;
   DATA[2060,9] := 2.0;
   DATA[2060,10] := 2.0;
   DATA[2060,11] := 19.76439;
   DATA[2060,12] := 2.209653;
   DATA[2060,13] := 802.799;
   DATA[2060,14] := 1.0;
   DATA[2060,15] := 2.0;
   DATA[2060,16] := 1.0;
   DATA[2060,17] := 1.0;
   DATA[2060,18] := 1.0;
   DATA[2060,19] := 2.0;
   DATA[2060,20] := 148.808;
   DATA[2060,21] := 154.8321;
   DATA[2060,22] := 1.719156;
   DATA[2060,23] := 834.0938;
   DATA[2060,24] := 2.0;
   DATA[2060,25] := 2.0;
   DATA[2060,26] := 7.874455;
   DATA[2060,27] := 143.9631;
   DATA[2060,28] := 262.0161;
   DATA[2060,29] := 12.07383;
   DATA[2060,30] := 1.730454;
   DATA[2060,31] := 1.297041;
   DATA[2060,32] := 0.7348846;
   DATA[2060,33] := 0.3068891;
   DATA[2060,34] := 2.0;
   DATA[2060,35] := 250.5928;
   DATA[2060,36] := 1.730048;
   DATA[2060,37] := 189.4386;
   DATA[2060,38] := 0.000128152;
   DATA[2060,39] := 1.0;
   DATA[2060,40] := 1.0;
   DATA[2061,0] := 2.461967;
   DATA[2061,1] := 861.284;
   DATA[2061,2] := 2.0;
   DATA[2061,3] := 2.0;
   DATA[2061,4] := 262.3686;
   DATA[2061,5] := 8.392271;
   DATA[2061,6] := 331.0946;
   DATA[2061,7] := 2.461667;
   DATA[2061,8] := 2.0;
   DATA[2061,9] := 2.0;
   DATA[2061,10] := 2.0;
   DATA[2061,11] := 19.76439;
   DATA[2061,12] := 2.207347;
   DATA[2061,13] := 802.8791;
   DATA[2061,14] := 1.0;
   DATA[2061,15] := 2.0;
   DATA[2061,16] := 1.0;
   DATA[2061,17] := 1.0;
   DATA[2061,18] := 1.0;
   DATA[2061,19] := 2.0;
   DATA[2061,20] := 148.808;
   DATA[2061,21] := 154.8321;
   DATA[2061,22] := 1.719156;
   DATA[2061,23] := 834.4399;
   DATA[2061,24] := 2.0;
   DATA[2061,25] := 2.0;
   DATA[2061,26] := 7.874455;
   DATA[2061,27] := 143.9631;
   DATA[2061,28] := 262.0161;
   DATA[2061,29] := 12.07383;
   DATA[2061,30] := 1.731479;
   DATA[2061,31] := 1.291533;
   DATA[2061,32] := 0.7348846;
   DATA[2061,33] := 0.3068891;
   DATA[2061,34] := 2.0;
   DATA[2061,35] := 250.5928;
   DATA[2061,36] := 1.730048;
   DATA[2061,37] := 189.4386;
   DATA[2061,38] := 0.000128152;
   DATA[2061,39] := 1.0;
   DATA[2061,40] := 1.0;
   DATA[2062,0] := 2.450437;
   DATA[2062,1] := 861.2055;
   DATA[2062,2] := 2.0;
   DATA[2062,3] := 2.0;
   DATA[2062,4] := 262.3686;
   DATA[2062,5] := 8.392271;
   DATA[2062,6] := 331.0946;
   DATA[2062,7] := 2.461667;
   DATA[2062,8] := 2.0;
   DATA[2062,9] := 2.0;
   DATA[2062,10] := 2.0;
   DATA[2062,11] := 19.76759;
   DATA[2062,12] := 2.206835;
   DATA[2062,13] := 802.9592;
   DATA[2062,14] := 1.0;
   DATA[2062,15] := 2.0;
   DATA[2062,16] := 1.0;
   DATA[2062,17] := 1.0;
   DATA[2062,18] := 1.0;
   DATA[2062,19] := 2.0;
   DATA[2062,20] := 148.808;
   DATA[2062,21] := 154.8321;
   DATA[2062,22] := 1.720053;
   DATA[2062,23] := 834.5937;
   DATA[2062,24] := 2.0;
   DATA[2062,25] := 2.0;
   DATA[2062,26] := 7.874455;
   DATA[2062,27] := 144.1169;
   DATA[2062,28] := 262.0161;
   DATA[2062,29] := 12.07383;
   DATA[2062,30] := 1.731479;
   DATA[2062,31] := 1.291277;
   DATA[2062,32] := 0.7348846;
   DATA[2062,33] := 0.306761;
   DATA[2062,34] := 2.0;
   DATA[2062,35] := 250.5928;
   DATA[2062,36] := 1.730048;
   DATA[2062,37] := 189.4386;
   DATA[2062,38] := 0.000128152;
   DATA[2062,39] := 1.0;
   DATA[2062,40] := 1.0;
   DATA[2063,0] := 2.437626;
   DATA[2063,1] := 861.5195;
   DATA[2063,2] := 2.0;
   DATA[2063,3] := 2.0;
   DATA[2063,4] := 262.3686;
   DATA[2063,5] := 8.392271;
   DATA[2063,6] := 331.0946;
   DATA[2063,7] := 2.46077;
   DATA[2063,8] := 2.0;
   DATA[2063,9] := 2.0;
   DATA[2063,10] := 2.0;
   DATA[2063,11] := 19.76759;
   DATA[2063,12] := 2.204913;
   DATA[2063,13] := 803.1194;
   DATA[2063,14] := 1.0;
   DATA[2063,15] := 2.0;
   DATA[2063,16] := 1.0;
   DATA[2063,17] := 1.0;
   DATA[2063,18] := 1.0;
   DATA[2063,19] := 2.0;
   DATA[2063,20] := 148.808;
   DATA[2063,21] := 154.8321;
   DATA[2063,22] := 1.720053;
   DATA[2063,23] := 834.5168;
   DATA[2063,24] := 2.0;
   DATA[2063,25] := 2.0;
   DATA[2063,26] := 7.874455;
   DATA[2063,27] := 144.1169;
   DATA[2063,28] := 262.0161;
   DATA[2063,29] := 11.76621;
   DATA[2063,30] := 1.73071;
   DATA[2063,31] := 1.283592;
   DATA[2063,32] := 0.7348846;
   DATA[2063,33] := 0.306761;
   DATA[2063,34] := 2.0;
   DATA[2063,35] := 250.5928;
   DATA[2063,36] := 1.730048;
   DATA[2063,37] := 189.4386;
   DATA[2063,38] := 0.000128152;
   DATA[2063,39] := 1.0;
   DATA[2063,40] := 1.0;
   DATA[2064,0] := 2.426737;
   DATA[2064,1] := 861.4803;
   DATA[2064,2] := 2.0;
   DATA[2064,3] := 2.0;
   DATA[2064,4] := 262.3686;
   DATA[2064,5] := 8.392271;
   DATA[2064,6] := 331.0946;
   DATA[2064,7] := 2.460257;
   DATA[2064,8] := 2.0;
   DATA[2064,9] := 2.0;
   DATA[2064,10] := 2.0;
   DATA[2064,11] := 19.72277;
   DATA[2064,12] := 2.204913;
   DATA[2064,13] := 803.56;
   DATA[2064,14] := 1.0;
   DATA[2064,15] := 2.0;
   DATA[2064,16] := 1.0;
   DATA[2064,17] := 1.0;
   DATA[2064,18] := 1.0;
   DATA[2064,19] := 2.0;
   DATA[2064,20] := 148.808;
   DATA[2064,21] := 154.8321;
   DATA[2064,22] := 1.720053;
   DATA[2064,23] := 834.4399;
   DATA[2064,24] := 2.0;
   DATA[2064,25] := 2.0;
   DATA[2064,26] := 7.874455;
   DATA[2064,27] := 144.1169;
   DATA[2064,28] := 262.0161;
   DATA[2064,29] := 11.76621;
   DATA[2064,30] := 1.728531;
   DATA[2064,31] := 1.287306;
   DATA[2064,32] := 0.7348846;
   DATA[2064,33] := 0.306761;
   DATA[2064,34] := 2.0;
   DATA[2064,35] := 250.7049;
   DATA[2064,36] := 1.730048;
   DATA[2064,37] := 189.4386;
   DATA[2064,38] := 0.000128152;
   DATA[2064,39] := 1.0;
   DATA[2064,40] := 1.0;
   DATA[2065,0] := 2.424815;
   DATA[2065,1] := 861.6765;
   DATA[2065,2] := 2.0;
   DATA[2065,3] := 2.0;
   DATA[2065,4] := 262.3686;
   DATA[2065,5] := 8.392271;
   DATA[2065,6] := 331.0946;
   DATA[2065,7] := 2.460257;
   DATA[2065,8] := 2.0;
   DATA[2065,9] := 2.0;
   DATA[2065,10] := 2.0;
   DATA[2065,11] := 19.72277;
   DATA[2065,12] := 2.204913;
   DATA[2065,13] := 803.4799;
   DATA[2065,14] := 1.0;
   DATA[2065,15] := 2.0;
   DATA[2065,16] := 1.0;
   DATA[2065,17] := 1.0;
   DATA[2065,18] := 1.0;
   DATA[2065,19] := 2.0;
   DATA[2065,20] := 148.808;
   DATA[2065,21] := 154.9603;
   DATA[2065,22] := 1.720053;
   DATA[2065,23] := 834.0554;
   DATA[2065,24] := 2.0;
   DATA[2065,25] := 2.0;
   DATA[2065,26] := 7.874455;
   DATA[2065,27] := 144.1169;
   DATA[2065,28] := 262.0161;
   DATA[2065,29] := 11.76621;
   DATA[2065,30] := 1.728531;
   DATA[2065,31] := 1.291277;
   DATA[2065,32] := 0.7348846;
   DATA[2065,33] := 0.3083624;
   DATA[2065,34] := 2.0;
   DATA[2065,35] := 250.8011;
   DATA[2065,36] := 1.730048;
   DATA[2065,37] := 189.4386;
   DATA[2065,38] := 0.000128152;
   DATA[2065,39] := 1.0;
   DATA[2065,40] := 1.0;
   DATA[2066,0] := 2.424815;
   DATA[2066,1] := 861.912;
   DATA[2066,2] := 2.0;
   DATA[2066,3] := 2.0;
   DATA[2066,4] := 262.3686;
   DATA[2066,5] := 8.392271;
   DATA[2066,6] := 331.0946;
   DATA[2066,7] := 2.460257;
   DATA[2066,8] := 2.0;
   DATA[2066,9] := 2.0;
   DATA[2066,10] := 2.0;
   DATA[2066,11] := 19.72277;
   DATA[2066,12] := 2.204913;
   DATA[2066,13] := 804.0006;
   DATA[2066,14] := 1.0;
   DATA[2066,15] := 2.0;
   DATA[2066,16] := 1.0;
   DATA[2066,17] := 1.0;
   DATA[2066,18] := 1.0;
   DATA[2066,19] := 2.0;
   DATA[2066,20] := 148.808;
   DATA[2066,21] := 154.9603;
   DATA[2066,22] := 1.718643;
   DATA[2066,23] := 833.7093;
   DATA[2066,24] := 2.0;
   DATA[2066,25] := 2.0;
   DATA[2066,26] := 7.874455;
   DATA[2066,27] := 144.1169;
   DATA[2066,28] := 262.0161;
   DATA[2066,29] := 12.07383;
   DATA[2066,30] := 1.728531;
   DATA[2066,31] := 1.291918;
   DATA[2066,32] := 0.7355248;
   DATA[2066,33] := 0.3086186;
   DATA[2066,34] := 2.0;
   DATA[2066,35] := 250.8011;
   DATA[2066,36] := 1.730048;
   DATA[2066,37] := 189.4546;
   DATA[2066,38] := 0.000128152;
   DATA[2066,39] := 1.0;
   DATA[2066,40] := 1.0;
   DATA[2067,0] := 2.462608;
   DATA[2067,1] := 862.3831;
   DATA[2067,2] := 2.0;
   DATA[2067,3] := 2.0;
   DATA[2067,4] := 262.3686;
   DATA[2067,5] := 8.392271;
   DATA[2067,6] := 331.0946;
   DATA[2067,7] := 2.458719;
   DATA[2067,8] := 2.0;
   DATA[2067,9] := 2.0;
   DATA[2067,10] := 2.0;
   DATA[2067,11] := 19.70997;
   DATA[2067,12] := 2.206707;
   DATA[2067,13] := 804.0006;
   DATA[2067,14] := 1.0;
   DATA[2067,15] := 2.0;
   DATA[2067,16] := 1.0;
   DATA[2067,17] := 1.0;
   DATA[2067,18] := 1.0;
   DATA[2067,19] := 2.0;
   DATA[2067,20] := 148.808;
   DATA[2067,21] := 154.9603;
   DATA[2067,22] := 1.71813;
   DATA[2067,23] := 833.8246;
   DATA[2067,24] := 2.0;
   DATA[2067,25] := 2.0;
   DATA[2067,26] := 7.874455;
   DATA[2067,27] := 144.0144;
   DATA[2067,28] := 262.0161;
   DATA[2067,29] := 12.07383;
   DATA[2067,30] := 1.728531;
   DATA[2067,31] := 1.301524;
   DATA[2067,32] := 0.7355248;
   DATA[2067,33] := 0.3086186;
   DATA[2067,34] := 2.0;
   DATA[2067,35] := 250.8011;
   DATA[2067,36] := 1.730048;
   DATA[2067,37] := 189.4546;
   DATA[2067,38] := 0.000128152;
   DATA[2067,39] := 1.0;
   DATA[2067,40] := 1.0;
   DATA[2068,0] := 2.509048;
   DATA[2068,1] := 862.7756;
   DATA[2068,2] := 2.0;
   DATA[2068,3] := 2.0;
   DATA[2068,4] := 262.3686;
   DATA[2068,5] := 8.392271;
   DATA[2068,6] := 331.0946;
   DATA[2068,7] := 2.457822;
   DATA[2068,8] := 2.0;
   DATA[2068,9] := 2.0;
   DATA[2068,10] := 2.0;
   DATA[2068,11] := 19.70997;
   DATA[2068,12] := 2.206963;
   DATA[2068,13] := 803.7603;
   DATA[2068,14] := 1.0;
   DATA[2068,15] := 2.0;
   DATA[2068,16] := 1.0;
   DATA[2068,17] := 1.0;
   DATA[2068,18] := 1.0;
   DATA[2068,19] := 2.0;
   DATA[2068,20] := 148.808;
   DATA[2068,21] := 154.9603;
   DATA[2068,22] := 1.71813;
   DATA[2068,23] := 833.7477;
   DATA[2068,24] := 2.0;
   DATA[2068,25] := 2.0;
   DATA[2068,26] := 7.874455;
   DATA[2068,27] := 143.9375;
   DATA[2068,28] := 262.0161;
   DATA[2068,29] := 12.07383;
   DATA[2068,30] := 1.728531;
   DATA[2068,31] := 1.302421;
   DATA[2068,32] := 0.7355248;
   DATA[2068,33] := 0.3086186;
   DATA[2068,34] := 2.0;
   DATA[2068,35] := 250.8011;
   DATA[2068,36] := 1.730048;
   DATA[2068,37] := 189.4546;
   DATA[2068,38] := 0.000128152;
   DATA[2068,39] := 1.0;
   DATA[2068,40] := 1.0;
   DATA[2069,0] := 2.547161;
   DATA[2069,1] := 862.4224;
   DATA[2069,2] := 2.0;
   DATA[2069,3] := 2.0;
   DATA[2069,4] := 262.3686;
   DATA[2069,5] := 8.392271;
   DATA[2069,6] := 331.0946;
   DATA[2069,7] := 2.457822;
   DATA[2069,8] := 2.0;
   DATA[2069,9] := 2.0;
   DATA[2069,10] := 2.0;
   DATA[2069,11] := 19.70997;
   DATA[2069,12] := 2.208372;
   DATA[2069,13] := 803.7603;
   DATA[2069,14] := 1.0;
   DATA[2069,15] := 2.0;
   DATA[2069,16] := 1.0;
   DATA[2069,17] := 1.0;
   DATA[2069,18] := 1.0;
   DATA[2069,19] := 2.0;
   DATA[2069,20] := 148.808;
   DATA[2069,21] := 154.9603;
   DATA[2069,22] := 1.720053;
   DATA[2069,23] := 834.0169;
   DATA[2069,24] := 2.0;
   DATA[2069,25] := 2.0;
   DATA[2069,26] := 7.874455;
   DATA[2069,27] := 143.9375;
   DATA[2069,28] := 262.0161;
   DATA[2069,29] := 12.07383;
   DATA[2069,30] := 1.728531;
   DATA[2069,31] := 1.296401;
   DATA[2069,32] := 0.7355248;
   DATA[2069,33] := 0.3086186;
   DATA[2069,34] := 2.0;
   DATA[2069,35] := 250.7049;
   DATA[2069,36] := 1.730048;
   DATA[2069,37] := 189.4546;
   DATA[2069,38] := 0.000128152;
   DATA[2069,39] := 1.0;
   DATA[2069,40] := 1.0;
   DATA[2070,0] := 2.589757;
   DATA[2070,1] := 862.4616;
   DATA[2070,2] := 2.0;
   DATA[2070,3] := 2.0;
   DATA[2070,4] := 262.3686;
   DATA[2070,5] := 8.392271;
   DATA[2070,6] := 331.0946;
   DATA[2070,7] := 2.457822;
   DATA[2070,8] := 2.0;
   DATA[2070,9] := 2.0;
   DATA[2070,10] := 2.0;
   DATA[2070,11] := 19.70997;
   DATA[2070,12] := 2.209397;
   DATA[2070,13] := 803.7202;
   DATA[2070,14] := 1.0;
   DATA[2070,15] := 2.0;
   DATA[2070,16] := 1.0;
   DATA[2070,17] := 1.0;
   DATA[2070,18] := 1.0;
   DATA[2070,19] := 2.0;
   DATA[2070,20] := 148.808;
   DATA[2070,21] := 154.9603;
   DATA[2070,22] := 1.720053;
   DATA[2070,23] := 833.7477;
   DATA[2070,24] := 2.0;
   DATA[2070,25] := 2.0;
   DATA[2070,26] := 7.874455;
   DATA[2070,27] := 143.9375;
   DATA[2070,28] := 262.0161;
   DATA[2070,29] := 12.03538;
   DATA[2070,30] := 1.728531;
   DATA[2070,31] := 1.281927;
   DATA[2070,32] := 0.7355248;
   DATA[2070,33] := 0.3086186;
   DATA[2070,34] := 2.0;
   DATA[2070,35] := 250.5768;
   DATA[2070,36] := 1.730048;
   DATA[2070,37] := 189.4546;
   DATA[2070,38] := 0.000128152;
   DATA[2070,39] := 1.0;
   DATA[2070,40] := 1.0;
   DATA[2071,0] := 2.626589;
   DATA[2071,1] := 862.4224;
   DATA[2071,2] := 2.0;
   DATA[2071,3] := 2.0;
   DATA[2071,4] := 262.3686;
   DATA[2071,5] := 8.392271;
   DATA[2071,6] := 331.0946;
   DATA[2071,7] := 2.460385;
   DATA[2071,8] := 2.0;
   DATA[2071,9] := 2.0;
   DATA[2071,10] := 2.0;
   DATA[2071,11] := 19.70997;
   DATA[2071,12] := 2.211575;
   DATA[2071,13] := 803.8004;
   DATA[2071,14] := 1.0;
   DATA[2071,15] := 2.0;
   DATA[2071,16] := 1.0;
   DATA[2071,17] := 1.0;
   DATA[2071,18] := 1.0;
   DATA[2071,19] := 2.0;
   DATA[2071,20] := 148.808;
   DATA[2071,21] := 154.9603;
   DATA[2071,22] := 1.720053;
   DATA[2071,23] := 833.517;
   DATA[2071,24] := 2.0;
   DATA[2071,25] := 2.0;
   DATA[2071,26] := 7.874455;
   DATA[2071,27] := 143.9375;
   DATA[2071,28] := 262.0161;
   DATA[2071,29] := 11.88157;
   DATA[2071,30] := 1.728531;
   DATA[2071,31] := 1.28167;
   DATA[2071,32] := 0.7355248;
   DATA[2071,33] := 0.3086186;
   DATA[2071,34] := 2.0;
   DATA[2071,35] := 250.5768;
   DATA[2071,36] := 1.730048;
   DATA[2071,37] := 189.4546;
   DATA[2071,38] := 0.000128152;
   DATA[2071,39] := 1.0;
   DATA[2071,40] := 1.0;
   DATA[2072,0] := 2.648048;
   DATA[2072,1] := 862.4616;
   DATA[2072,2] := 2.0;
   DATA[2072,3] := 2.0;
   DATA[2072,4] := 262.3686;
   DATA[2072,5] := 8.392271;
   DATA[2072,6] := 331.0946;
   DATA[2072,7] := 2.460385;
   DATA[2072,8] := 2.0;
   DATA[2072,9] := 2.0;
   DATA[2072,10] := 2.0;
   DATA[2072,11] := 19.65235;
   DATA[2072,12] := 2.212215;
   DATA[2072,13] := 803.56;
   DATA[2072,14] := 1.0;
   DATA[2072,15] := 2.0;
   DATA[2072,16] := 1.0;
   DATA[2072,17] := 1.0;
   DATA[2072,18] := 1.0;
   DATA[2072,19] := 2.0;
   DATA[2072,20] := 148.808;
   DATA[2072,21] := 154.9603;
   DATA[2072,22] := 1.719027;
   DATA[2072,23] := 833.3248;
   DATA[2072,24] := 2.0;
   DATA[2072,25] := 2.0;
   DATA[2072,26] := 7.874455;
   DATA[2072,27] := 143.9375;
   DATA[2072,28] := 262.0161;
   DATA[2072,29] := 11.88157;
   DATA[2072,30] := 1.728531;
   DATA[2072,31] := 1.28167;
   DATA[2072,32] := 0.7355248;
   DATA[2072,33] := 0.3086186;
   DATA[2072,34] := 2.0;
   DATA[2072,35] := 250.5768;
   DATA[2072,36] := 1.730048;
   DATA[2072,37] := 189.3425;
   DATA[2072,38] := 0.000128152;
   DATA[2072,39] := 1.0;
   DATA[2072,40] := 1.0;
   DATA[2073,0] := 2.657656;
   DATA[2073,1] := 862.5009;
   DATA[2073,2] := 2.0;
   DATA[2073,3] := 2.0;
   DATA[2073,4] := 262.3686;
   DATA[2073,5] := 8.392271;
   DATA[2073,6] := 331.0946;
   DATA[2073,7] := 2.460385;
   DATA[2073,8] := 2.0;
   DATA[2073,9] := 2.0;
   DATA[2073,10] := 2.0;
   DATA[2073,11] := 19.65235;
   DATA[2073,12] := 2.212215;
   DATA[2073,13] := 803.9205;
   DATA[2073,14] := 1.0;
   DATA[2073,15] := 2.0;
   DATA[2073,16] := 1.0;
   DATA[2073,17] := 1.0;
   DATA[2073,18] := 1.0;
   DATA[2073,19] := 2.0;
   DATA[2073,20] := 148.808;
   DATA[2073,21] := 154.9603;
   DATA[2073,22] := 1.717361;
   DATA[2073,23] := 833.4786;
   DATA[2073,24] := 2.0;
   DATA[2073,25] := 2.0;
   DATA[2073,26] := 7.874455;
   DATA[2073,27] := 143.9375;
   DATA[2073,28] := 262.0161;
   DATA[2073,29] := 11.88157;
   DATA[2073,30] := 1.7293;
   DATA[2073,31] := 1.28167;
   DATA[2073,32] := 0.7355248;
   DATA[2073,33] := 0.306761;
   DATA[2073,34] := 2.0;
   DATA[2073,35] := 250.5768;
   DATA[2073,36] := 1.730048;
   DATA[2073,37] := 189.3425;
   DATA[2073,38] := 0.000128152;
   DATA[2073,39] := 1.0;
   DATA[2073,40] := 1.0;
   DATA[2074,0] := 2.646446;
   DATA[2074,1] := 862.7756;
   DATA[2074,2] := 2.0;
   DATA[2074,3] := 2.0;
   DATA[2074,4] := 262.3686;
   DATA[2074,5] := 8.392271;
   DATA[2074,6] := 331.0946;
   DATA[2074,7] := 2.461667;
   DATA[2074,8] := 2.0;
   DATA[2074,9] := 2.0;
   DATA[2074,10] := 2.0;
   DATA[2074,11] := 19.66835;
   DATA[2074,12] := 2.2126;
   DATA[2074,13] := 803.6;
   DATA[2074,14] := 1.0;
   DATA[2074,15] := 2.0;
   DATA[2074,16] := 1.0;
   DATA[2074,17] := 1.0;
   DATA[2074,18] := 1.0;
   DATA[2074,19] := 2.0;
   DATA[2074,20] := 148.808;
   DATA[2074,21] := 154.9603;
   DATA[2074,22] := 1.717233;
   DATA[2074,23] := 833.5555;
   DATA[2074,24] := 2.0;
   DATA[2074,25] := 2.0;
   DATA[2074,26] := 7.874455;
   DATA[2074,27] := 143.9375;
   DATA[2074,28] := 262.0161;
   DATA[2074,29] := 11.88157;
   DATA[2074,30] := 1.730582;
   DATA[2074,31] := 1.294479;
   DATA[2074,32] := 0.7355248;
   DATA[2074,33] := 0.306761;
   DATA[2074,34] := 2.0;
   DATA[2074,35] := 250.5768;
   DATA[2074,36] := 1.730048;
   DATA[2074,37] := 189.3425;
   DATA[2074,38] := 0.000128152;
   DATA[2074,39] := 1.0;
   DATA[2074,40] := 1.0;
   DATA[2075,0] := 2.629152;
   DATA[2075,1] := 863.4037;
   DATA[2075,2] := 2.0;
   DATA[2075,3] := 2.0;
   DATA[2075,4] := 262.3686;
   DATA[2075,5] := 8.392271;
   DATA[2075,6] := 331.0946;
   DATA[2075,7] := 2.461667;
   DATA[2075,8] := 2.0;
   DATA[2075,9] := 2.0;
   DATA[2075,10] := 2.0;
   DATA[2075,11] := 19.74198;
   DATA[2075,12] := 2.2126;
   DATA[2075,13] := 803.7603;
   DATA[2075,14] := 1.0;
   DATA[2075,15] := 2.0;
   DATA[2075,16] := 1.0;
   DATA[2075,17] := 1.0;
   DATA[2075,18] := 1.0;
   DATA[2075,19] := 2.0;
   DATA[2075,20] := 148.808;
   DATA[2075,21] := 154.9603;
   DATA[2075,22] := 1.717233;
   DATA[2075,23] := 833.7477;
   DATA[2075,24] := 2.0;
   DATA[2075,25] := 2.0;
   DATA[2075,26] := 7.874455;
   DATA[2075,27] := 143.9375;
   DATA[2075,28] := 262.0161;
   DATA[2075,29] := 11.88157;
   DATA[2075,30] := 1.730582;
   DATA[2075,31] := 1.294479;
   DATA[2075,32] := 0.7355248;
   DATA[2075,33] := 0.306761;
   DATA[2075,34] := 2.0;
   DATA[2075,35] := 250.5768;
   DATA[2075,36] := 1.730048;
   DATA[2075,37] := 189.3425;
   DATA[2075,38] := 0.000128152;
   DATA[2075,39] := 1.0;
   DATA[2075,40] := 1.0;
   DATA[2076,0] := 2.614419;
   DATA[2076,1] := 863.757;
   DATA[2076,2] := 2.0;
   DATA[2076,3] := 2.0;
   DATA[2076,4] := 262.3686;
   DATA[2076,5] := 8.392271;
   DATA[2076,6] := 331.0946;
   DATA[2076,7] := 2.461667;
   DATA[2076,8] := 2.0;
   DATA[2076,9] := 2.0;
   DATA[2076,10] := 2.0;
   DATA[2076,11] := 19.74198;
   DATA[2076,12] := 2.2126;
   DATA[2076,13] := 803.9205;
   DATA[2076,14] := 1.0;
   DATA[2076,15] := 2.0;
   DATA[2076,16] := 1.0;
   DATA[2076,17] := 1.0;
   DATA[2076,18] := 1.0;
   DATA[2076,19] := 2.0;
   DATA[2076,20] := 148.808;
   DATA[2076,21] := 154.9603;
   DATA[2076,22] := 1.715824;
   DATA[2076,23] := 834.0938;
   DATA[2076,24] := 2.0;
   DATA[2076,25] := 2.0;
   DATA[2076,26] := 7.874455;
   DATA[2076,27] := 143.9375;
   DATA[2076,28] := 262.0161;
   DATA[2076,29] := 11.88157;
   DATA[2076,30] := 1.730582;
   DATA[2076,31] := 1.291789;
   DATA[2076,32] := 0.7355248;
   DATA[2076,33] := 0.306761;
   DATA[2076,34] := 2.0;
   DATA[2076,35] := 250.2724;
   DATA[2076,36] := 1.730048;
   DATA[2076,37] := 189.3425;
   DATA[2076,38] := 0.000128152;
   DATA[2076,39] := 1.0;
   DATA[2076,40] := 1.0;
   DATA[2077,0] := 2.607693;
   DATA[2077,1] := 863.8354;
   DATA[2077,2] := 2.0;
   DATA[2077,3] := 2.0;
   DATA[2077,4] := 262.3686;
   DATA[2077,5] := 8.392271;
   DATA[2077,6] := 331.0946;
   DATA[2077,7] := 2.458847;
   DATA[2077,8] := 2.0;
   DATA[2077,9] := 2.0;
   DATA[2077,10] := 2.0;
   DATA[2077,11] := 19.74198;
   DATA[2077,12] := 2.210166;
   DATA[2077,13] := 803.7202;
   DATA[2077,14] := 1.0;
   DATA[2077,15] := 2.0;
   DATA[2077,16] := 1.0;
   DATA[2077,17] := 1.0;
   DATA[2077,18] := 1.0;
   DATA[2077,19] := 2.0;
   DATA[2077,20] := 148.808;
   DATA[2077,21] := 154.9603;
   DATA[2077,22] := 1.715311;
   DATA[2077,23] := 834.4014;
   DATA[2077,24] := 2.0;
   DATA[2077,25] := 2.0;
   DATA[2077,26] := 7.874455;
   DATA[2077,27] := 143.9375;
   DATA[2077,28] := 262.0161;
   DATA[2077,29] := 12.07383;
   DATA[2077,30] := 1.730582;
   DATA[2077,31] := 1.294351;
   DATA[2077,32] := 0.7355248;
   DATA[2077,33] := 0.306761;
   DATA[2077,34] := 2.0;
   DATA[2077,35] := 250.2724;
   DATA[2077,36] := 1.730048;
   DATA[2077,37] := 189.1342;
   DATA[2077,38] := 0.000128152;
   DATA[2077,39] := 1.0;
   DATA[2077,40] := 1.0;
   DATA[2078,0] := 2.594882;
   DATA[2078,1] := 863.757;
   DATA[2078,2] := 2.0;
   DATA[2078,3] := 2.0;
   DATA[2078,4] := 262.3686;
   DATA[2078,5] := 8.392271;
   DATA[2078,6] := 331.0946;
   DATA[2078,7] := 2.458847;
   DATA[2078,8] := 2.0;
   DATA[2078,9] := 2.0;
   DATA[2078,10] := 2.0;
   DATA[2078,11] := 19.73558;
   DATA[2078,12] := 2.210166;
   DATA[2078,13] := 804.1207;
   DATA[2078,14] := 1.0;
   DATA[2078,15] := 2.0;
   DATA[2078,16] := 1.0;
   DATA[2078,17] := 1.0;
   DATA[2078,18] := 1.0;
   DATA[2078,19] := 2.0;
   DATA[2078,20] := 148.808;
   DATA[2078,21] := 154.9603;
   DATA[2078,22] := 1.715311;
   DATA[2078,23] := 835.0551;
   DATA[2078,24] := 2.0;
   DATA[2078,25] := 2.0;
   DATA[2078,26] := 7.874455;
   DATA[2078,27] := 143.9375;
   DATA[2078,28] := 262.0161;
   DATA[2078,29] := 12.07383;
   DATA[2078,30] := 1.72725;
   DATA[2078,31] := 1.302677;
   DATA[2078,32] := 0.7355248;
   DATA[2078,33] := 0.3081062;
   DATA[2078,34] := 2.0;
   DATA[2078,35] := 250.2243;
   DATA[2078,36] := 1.730048;
   DATA[2078,37] := 189.1022;
   DATA[2078,38] := 0.000128152;
   DATA[2078,39] := 1.0;
   DATA[2078,40] := 1.0;
   DATA[2079,0] := 2.577587;
   DATA[2079,1] := 863.9532;
   DATA[2079,2] := 2.0;
   DATA[2079,3] := 2.0;
   DATA[2079,4] := 262.3686;
   DATA[2079,5] := 8.392271;
   DATA[2079,6] := 331.0946;
   DATA[2079,7] := 2.458847;
   DATA[2079,8] := 2.0;
   DATA[2079,9] := 2.0;
   DATA[2079,10] := 2.0;
   DATA[2079,11] := 19.73558;
   DATA[2079,12] := 2.207988;
   DATA[2079,13] := 804.0807;
   DATA[2079,14] := 1.0;
   DATA[2079,15] := 2.0;
   DATA[2079,16] := 1.0;
   DATA[2079,17] := 1.0;
   DATA[2079,18] := 1.0;
   DATA[2079,19] := 2.0;
   DATA[2079,20] := 148.808;
   DATA[2079,21] := 154.9603;
   DATA[2079,22] := 1.715311;
   DATA[2079,23] := 835.0936;
   DATA[2079,24] := 2.0;
   DATA[2079,25] := 2.0;
   DATA[2079,26] := 7.874455;
   DATA[2079,27] := 143.9375;
   DATA[2079,28] := 262.0161;
   DATA[2079,29] := 12.07383;
   DATA[2079,30] := 1.726865;
   DATA[2079,31] := 1.293455;
   DATA[2079,32] := 0.7355248;
   DATA[2079,33] := 0.3086186;
   DATA[2079,34] := 2.0;
   DATA[2079,35] := 250.2243;
   DATA[2079,36] := 1.730048;
   DATA[2079,37] := 189.0381;
   DATA[2079,38] := 0.000128152;
   DATA[2079,39] := 1.0;
   DATA[2079,40] := 1.0;
   DATA[2080,0] := 2.559331;
   DATA[2080,1] := 863.5999;
   DATA[2080,2] := 2.0;
   DATA[2080,3] := 2.0;
   DATA[2080,4] := 262.3686;
   DATA[2080,5] := 8.392271;
   DATA[2080,6] := 331.0946;
   DATA[2080,7] := 2.460001;
   DATA[2080,8] := 2.0;
   DATA[2080,9] := 2.0;
   DATA[2080,10] := 2.0;
   DATA[2080,11] := 19.73558;
   DATA[2080,12] := 2.206194;
   DATA[2080,13] := 803.9606;
   DATA[2080,14] := 1.0;
   DATA[2080,15] := 2.0;
   DATA[2080,16] := 1.0;
   DATA[2080,17] := 1.0;
   DATA[2080,18] := 1.0;
   DATA[2080,19] := 2.0;
   DATA[2080,20] := 148.808;
   DATA[2080,21] := 154.9603;
   DATA[2080,22] := 1.715311;
   DATA[2080,23] := 835.2858;
   DATA[2080,24] := 2.0;
   DATA[2080,25] := 2.0;
   DATA[2080,26] := 7.874455;
   DATA[2080,27] := 143.9375;
   DATA[2080,28] := 262.0161;
   DATA[2080,29] := 12.07383;
   DATA[2080,30] := 1.726865;
   DATA[2080,31] := 1.29781;
   DATA[2080,32] := 0.7355248;
   DATA[2080,33] := 0.3086186;
   DATA[2080,34] := 2.0;
   DATA[2080,35] := 250.2243;
   DATA[2080,36] := 1.730048;
   DATA[2080,37] := 189.0381;
   DATA[2080,38] := 0.000128152;
   DATA[2080,39] := 1.0;
   DATA[2080,40] := 1.0;
   DATA[2081,0] := 2.540435;
   DATA[2081,1] := 863.9924;
   DATA[2081,2] := 2.0;
   DATA[2081,3] := 2.0;
   DATA[2081,4] := 262.3686;
   DATA[2081,5] := 8.392271;
   DATA[2081,6] := 331.0946;
   DATA[2081,7] := 2.460385;
   DATA[2081,8] := 2.0;
   DATA[2081,9] := 2.0;
   DATA[2081,10] := 2.0;
   DATA[2081,11] := 19.76759;
   DATA[2081,12] := 2.206194;
   DATA[2081,13] := 804.2009;
   DATA[2081,14] := 1.0;
   DATA[2081,15] := 2.0;
   DATA[2081,16] := 1.0;
   DATA[2081,17] := 1.0;
   DATA[2081,18] := 1.0;
   DATA[2081,19] := 2.0;
   DATA[2081,20] := 148.808;
   DATA[2081,21] := 154.9603;
   DATA[2081,22] := 1.717489;
   DATA[2081,23] := 835.4396;
   DATA[2081,24] := 2.0;
   DATA[2081,25] := 2.0;
   DATA[2081,26] := 7.874455;
   DATA[2081,27] := 143.9375;
   DATA[2081,28] := 262.0161;
   DATA[2081,29] := 12.07383;
   DATA[2081,30] := 1.726865;
   DATA[2081,31] := 1.291533;
   DATA[2081,32] := 0.7355248;
   DATA[2081,33] := 0.3086186;
   DATA[2081,34] := 2.0;
   DATA[2081,35] := 250.2243;
   DATA[2081,36] := 1.730048;
   DATA[2081,37] := 189.0381;
   DATA[2081,38] := 0.000128152;
   DATA[2081,39] := 1.0;
   DATA[2081,40] := 1.0;
   DATA[2082,0] := 2.520898;
   DATA[2082,1] := 864.071;
   DATA[2082,2] := 2.0;
   DATA[2082,3] := 2.0;
   DATA[2082,4] := 262.1443;
   DATA[2082,5] := 8.392271;
   DATA[2082,6] := 331.0946;
   DATA[2082,7] := 2.460385;
   DATA[2082,8] := 2.0;
   DATA[2082,9] := 2.0;
   DATA[2082,10] := 2.0;
   DATA[2082,11] := 19.76759;
   DATA[2082,12] := 2.206194;
   DATA[2082,13] := 804.0807;
   DATA[2082,14] := 1.0;
   DATA[2082,15] := 2.0;
   DATA[2082,16] := 1.0;
   DATA[2082,17] := 1.0;
   DATA[2082,18] := 1.0;
   DATA[2082,19] := 2.0;
   DATA[2082,20] := 148.808;
   DATA[2082,21] := 154.9603;
   DATA[2082,22] := 1.717746;
   DATA[2082,23] := 835.8626;
   DATA[2082,24] := 2.0;
   DATA[2082,25] := 2.0;
   DATA[2082,26] := 7.874455;
   DATA[2082,27] := 143.9375;
   DATA[2082,28] := 262.0161;
   DATA[2082,29] := 12.07383;
   DATA[2082,30] := 1.726865;
   DATA[2082,31] := 1.281927;
   DATA[2082,32] := 0.7355248;
   DATA[2082,33] := 0.3086186;
   DATA[2082,34] := 2.0;
   DATA[2082,35] := 250.2243;
   DATA[2082,36] := 1.730048;
   DATA[2082,37] := 189.0381;
   DATA[2082,38] := 0.000128152;
   DATA[2082,39] := 1.0;
   DATA[2082,40] := 1.0;
   DATA[2083,0] := 2.505845;
   DATA[2083,1] := 864.1495;
   DATA[2083,2] := 2.0;
   DATA[2083,3] := 2.0;
   DATA[2083,4] := 262.1443;
   DATA[2083,5] := 8.392271;
   DATA[2083,6] := 330.9408;
   DATA[2083,7] := 2.460385;
   DATA[2083,8] := 2.0;
   DATA[2083,9] := 2.0;
   DATA[2083,10] := 2.0;
   DATA[2083,11] := 19.72598;
   DATA[2083,12] := 2.208628;
   DATA[2083,13] := 804.2809;
   DATA[2083,14] := 1.0;
   DATA[2083,15] := 2.0;
   DATA[2083,16] := 1.0;
   DATA[2083,17] := 1.0;
   DATA[2083,18] := 1.0;
   DATA[2083,19] := 2.0;
   DATA[2083,20] := 148.808;
   DATA[2083,21] := 154.9603;
   DATA[2083,22] := 1.717746;
   DATA[2083,23] := 835.9395;
   DATA[2083,24] := 2.0;
   DATA[2083,25] := 2.0;
   DATA[2083,26] := 7.874455;
   DATA[2083,27] := 143.9375;
   DATA[2083,28] := 262.0161;
   DATA[2083,29] := 12.07383;
   DATA[2083,30] := 1.726865;
   DATA[2083,31] := 1.289612;
   DATA[2083,32] := 0.7355248;
   DATA[2083,33] := 0.3086186;
   DATA[2083,34] := 2.0;
   DATA[2083,35] := 250.3044;
   DATA[2083,36] := 1.730048;
   DATA[2083,37] := 189.0541;
   DATA[2083,38] := 0.000128152;
   DATA[2083,39] := 1.0;
   DATA[2083,40] := 1.0;
   DATA[2084,0] := 2.491432;
   DATA[2084,1] := 863.9532;
   DATA[2084,2] := 2.0;
   DATA[2084,3] := 2.0;
   DATA[2084,4] := 262.1443;
   DATA[2084,5] := 8.392271;
   DATA[2084,6] := 330.8639;
   DATA[2084,7] := 2.460385;
   DATA[2084,8] := 2.0;
   DATA[2084,9] := 2.0;
   DATA[2084,10] := 2.0;
   DATA[2084,11] := 19.72598;
   DATA[2084,12] := 2.208628;
   DATA[2084,13] := 804.5613;
   DATA[2084,14] := 1.0;
   DATA[2084,15] := 2.0;
   DATA[2084,16] := 1.0;
   DATA[2084,17] := 1.0;
   DATA[2084,18] := 1.0;
   DATA[2084,19] := 2.0;
   DATA[2084,20] := 148.808;
   DATA[2084,21] := 154.9603;
   DATA[2084,22] := 1.721334;
   DATA[2084,23] := 835.7857;
   DATA[2084,24] := 2.0;
   DATA[2084,25] := 2.0;
   DATA[2084,26] := 7.874455;
   DATA[2084,27] := 143.9375;
   DATA[2084,28] := 262.0161;
   DATA[2084,29] := 12.07383;
   DATA[2084,30] := 1.7293;
   DATA[2084,31] := 1.292558;
   DATA[2084,32] := 0.7355248;
   DATA[2084,33] := 0.3086186;
   DATA[2084,34] := 2.0;
   DATA[2084,35] := 250.3365;
   DATA[2084,36] := 1.730048;
   DATA[2084,37] := 189.2143;
   DATA[2084,38] := 0.000128152;
   DATA[2084,39] := 1.0;
   DATA[2084,40] := 1.0;
   DATA[2085,0] := 2.4767;
   DATA[2085,1] := 863.9924;
   DATA[2085,2] := 2.0;
   DATA[2085,3] := 2.0;
   DATA[2085,4] := 262.3686;
   DATA[2085,5] := 8.392271;
   DATA[2085,6] := 330.8639;
   DATA[2085,7] := 2.460385;
   DATA[2085,8] := 2.0;
   DATA[2085,9] := 2.0;
   DATA[2085,10] := 2.0;
   DATA[2085,11] := 19.72598;
   DATA[2085,12] := 2.208628;
   DATA[2085,13] := 804.5213;
   DATA[2085,14] := 1.0;
   DATA[2085,15] := 2.0;
   DATA[2085,16] := 1.0;
   DATA[2085,17] := 1.0;
   DATA[2085,18] := 1.0;
   DATA[2085,19] := 2.0;
   DATA[2085,20] := 148.808;
   DATA[2085,21] := 154.9603;
   DATA[2085,22] := 1.721334;
   DATA[2085,23] := 836.3625;
   DATA[2085,24] := 2.0;
   DATA[2085,25] := 2.0;
   DATA[2085,26] := 7.874455;
   DATA[2085,27] := 143.9887;
   DATA[2085,28] := 262.0161;
   DATA[2085,29] := 12.07383;
   DATA[2085,30] := 1.7293;
   DATA[2085,31] := 1.292558;
   DATA[2085,32] := 0.7355248;
   DATA[2085,33] := 0.3086186;
   DATA[2085,34] := 2.0;
   DATA[2085,35] := 250.3845;
   DATA[2085,36] := 1.730048;
   DATA[2085,37] := 189.2143;
   DATA[2085,38] := 0.000128152;
   DATA[2085,39] := 1.0;
   DATA[2085,40] := 1.0;
   DATA[2086,0] := 2.464209;
   DATA[2086,1] := 864.2672;
   DATA[2086,2] := 2.0;
   DATA[2086,3] := 2.0;
   DATA[2086,4] := 262.4007;
   DATA[2086,5] := 8.392271;
   DATA[2086,6] := 330.8639;
   DATA[2086,7] := 2.460385;
   DATA[2086,8] := 2.0;
   DATA[2086,9] := 2.0;
   DATA[2086,10] := 2.0;
   DATA[2086,11] := 19.72598;
   DATA[2086,12] := 2.208628;
   DATA[2086,13] := 805.3224;
   DATA[2086,14] := 1.0;
   DATA[2086,15] := 2.0;
   DATA[2086,16] := 1.0;
   DATA[2086,17] := 1.0;
   DATA[2086,18] := 1.0;
   DATA[2086,19] := 2.0;
   DATA[2086,20] := 148.808;
   DATA[2086,21] := 154.9603;
   DATA[2086,22] := 1.721334;
   DATA[2086,23] := 836.6317;
   DATA[2086,24] := 2.0;
   DATA[2086,25] := 2.0;
   DATA[2086,26] := 7.874455;
   DATA[2086,27] := 144.0656;
   DATA[2086,28] := 262.0161;
   DATA[2086,29] := 12.07383;
   DATA[2086,30] := 1.7293;
   DATA[2086,31] := 1.292558;
   DATA[2086,32] := 0.7355248;
   DATA[2086,33] := 0.3077219;
   DATA[2086,34] := 2.0;
   DATA[2086,35] := 250.3845;
   DATA[2086,36] := 1.730048;
   DATA[2086,37] := 189.2143;
   DATA[2086,38] := 0.000128152;
   DATA[2086,39] := 1.0;
   DATA[2086,40] := 1.0;
   DATA[2087,0] := 2.450758;
   DATA[2087,1] := 863.7962;
   DATA[2087,2] := 2.0;
   DATA[2087,3] := 2.0;
   DATA[2087,4] := 262.4007;
   DATA[2087,5] := 8.392271;
   DATA[2087,6] := 330.8639;
   DATA[2087,7] := 2.460385;
   DATA[2087,8] := 2.0;
   DATA[2087,9] := 2.0;
   DATA[2087,10] := 2.0;
   DATA[2087,11] := 19.70357;
   DATA[2087,12] := 2.208628;
   DATA[2087,13] := 805.6027;
   DATA[2087,14] := 1.0;
   DATA[2087,15] := 2.0;
   DATA[2087,16] := 1.0;
   DATA[2087,17] := 1.0;
   DATA[2087,18] := 1.0;
   DATA[2087,19] := 2.0;
   DATA[2087,20] := 148.808;
   DATA[2087,21] := 154.9603;
   DATA[2087,22] := 1.719668;
   DATA[2087,23] := 836.3625;
   DATA[2087,24] := 2.0;
   DATA[2087,25] := 2.0;
   DATA[2087,26] := 7.874455;
   DATA[2087,27] := 144.0656;
   DATA[2087,28] := 262.0161;
   DATA[2087,29] := 12.07383;
   DATA[2087,30] := 1.72725;
   DATA[2087,31] := 1.292558;
   DATA[2087,32] := 0.7355248;
   DATA[2087,33] := 0.3065689;
   DATA[2087,34] := 2.0;
   DATA[2087,35] := 250.3845;
   DATA[2087,36] := 1.730048;
   DATA[2087,37] := 189.2143;
   DATA[2087,38] := 0.000128152;
   DATA[2087,39] := 1.0;
   DATA[2087,40] := 1.0;
   DATA[2088,0] := 2.434744;
   DATA[2088,1] := 864.0317;
   DATA[2088,2] := 2.0;
   DATA[2088,3] := 2.0;
   DATA[2088,4] := 262.4007;
   DATA[2088,5] := 8.392271;
   DATA[2088,6] := 330.8639;
   DATA[2088,7] := 2.460385;
   DATA[2088,8] := 2.0;
   DATA[2088,9] := 2.0;
   DATA[2088,10] := 2.0;
   DATA[2088,11] := 19.70357;
   DATA[2088,12] := 2.208628;
   DATA[2088,13] := 805.5627;
   DATA[2088,14] := 1.0;
   DATA[2088,15] := 2.0;
   DATA[2088,16] := 1.0;
   DATA[2088,17] := 1.0;
   DATA[2088,18] := 1.0;
   DATA[2088,19] := 2.0;
   DATA[2088,20] := 148.808;
   DATA[2088,21] := 154.9603;
   DATA[2088,22] := 1.718771;
   DATA[2088,23] := 836.7086;
   DATA[2088,24] := 2.0;
   DATA[2088,25] := 2.0;
   DATA[2088,26] := 7.874455;
   DATA[2088,27] := 144.0656;
   DATA[2088,28] := 262.0161;
   DATA[2088,29] := 12.07383;
   DATA[2088,30] := 1.72725;
   DATA[2088,31] := 1.292174;
   DATA[2088,32] := 0.7355248;
   DATA[2088,33] := 0.3065689;
   DATA[2088,34] := 2.0;
   DATA[2088,35] := 250.3845;
   DATA[2088,36] := 1.730048;
   DATA[2088,37] := 189.2143;
   DATA[2088,38] := 0.000128152;
   DATA[2088,39] := 1.0;
   DATA[2088,40] := 1.0;
   DATA[2089,0] := 2.428338;
   DATA[2089,1] := 863.2466;
   DATA[2089,2] := 2.0;
   DATA[2089,3] := 2.0;
   DATA[2089,4] := 262.4007;
   DATA[2089,5] := 8.392271;
   DATA[2089,6] := 330.8639;
   DATA[2089,7] := 2.457694;
   DATA[2089,8] := 2.0;
   DATA[2089,9] := 2.0;
   DATA[2089,10] := 2.0;
   DATA[2089,11] := 19.76759;
   DATA[2089,12] := 2.208628;
   DATA[2089,13] := 805.7229;
   DATA[2089,14] := 1.0;
   DATA[2089,15] := 2.0;
   DATA[2089,16] := 1.0;
   DATA[2089,17] := 1.0;
   DATA[2089,18] := 1.0;
   DATA[2089,19] := 2.0;
   DATA[2089,20] := 148.808;
   DATA[2089,21] := 154.9603;
   DATA[2089,22] := 1.718771;
   DATA[2089,23] := 836.5932;
   DATA[2089,24] := 2.0;
   DATA[2089,25] := 2.0;
   DATA[2089,26] := 7.874455;
   DATA[2089,27] := 144.0656;
   DATA[2089,28] := 262.0161;
   DATA[2089,29] := 12.07383;
   DATA[2089,30] := 1.724942;
   DATA[2089,31] := 1.298322;
   DATA[2089,32] := 0.7355248;
   DATA[2089,33] := 0.3065689;
   DATA[2089,34] := 2.0;
   DATA[2089,35] := 250.3845;
   DATA[2089,36] := 1.730048;
   DATA[2089,37] := 189.2143;
   DATA[2089,38] := 0.000128152;
   DATA[2089,39] := 1.0;
   DATA[2089,40] := 1.0;
   DATA[2090,0] := 2.428018;
   DATA[2090,1] := 863.1682;
   DATA[2090,2] := 2.0;
   DATA[2090,3] := 2.0;
   DATA[2090,4] := 262.4007;
   DATA[2090,5] := 8.392271;
   DATA[2090,6] := 330.8639;
   DATA[2090,7] := 2.457694;
   DATA[2090,8] := 2.0;
   DATA[2090,9] := 2.0;
   DATA[2090,10] := 2.0;
   DATA[2090,11] := 19.77079;
   DATA[2090,12] := 2.209909;
   DATA[2090,13] := 805.6829;
   DATA[2090,14] := 1.0;
   DATA[2090,15] := 2.0;
   DATA[2090,16] := 1.0;
   DATA[2090,17] := 1.0;
   DATA[2090,18] := 1.0;
   DATA[2090,19] := 2.0;
   DATA[2090,20] := 148.808;
   DATA[2090,21] := 154.9603;
   DATA[2090,22] := 1.718771;
   DATA[2090,23] := 836.4394;
   DATA[2090,24] := 2.0;
   DATA[2090,25] := 2.0;
   DATA[2090,26] := 7.874455;
   DATA[2090,27] := 144.0656;
   DATA[2090,28] := 262.0161;
   DATA[2090,29] := 12.07383;
   DATA[2090,30] := 1.724686;
   DATA[2090,31] := 1.28705;
   DATA[2090,32] := 0.7355248;
   DATA[2090,33] := 0.3065689;
   DATA[2090,34] := 2.0;
   DATA[2090,35] := 250.3845;
   DATA[2090,36] := 1.730048;
   DATA[2090,37] := 189.1182;
   DATA[2090,38] := 0.000128152;
   DATA[2090,39] := 1.0;
   DATA[2090,40] := 1.0;
   DATA[2091,0] := 2.428018;
   DATA[2091,1] := 863.0897;
   DATA[2091,2] := 2.0;
   DATA[2091,3] := 2.0;
   DATA[2091,4] := 262.4007;
   DATA[2091,5] := 8.392271;
   DATA[2091,6] := 330.8639;
   DATA[2091,7] := 2.457694;
   DATA[2091,8] := 2.0;
   DATA[2091,9] := 2.0;
   DATA[2091,10] := 2.0;
   DATA[2091,11] := 19.77079;
   DATA[2091,12] := 2.209909;
   DATA[2091,13] := 805.9633;
   DATA[2091,14] := 1.0;
   DATA[2091,15] := 2.0;
   DATA[2091,16] := 1.0;
   DATA[2091,17] := 1.0;
   DATA[2091,18] := 1.0;
   DATA[2091,19] := 2.0;
   DATA[2091,20] := 148.808;
   DATA[2091,21] := 155.0115;
   DATA[2091,22] := 1.718771;
   DATA[2091,23] := 836.2087;
   DATA[2091,24] := 2.0;
   DATA[2091,25] := 2.0;
   DATA[2091,26] := 7.874455;
   DATA[2091,27] := 144.0656;
   DATA[2091,28] := 262.0161;
   DATA[2091,29] := 12.07383;
   DATA[2091,30] := 1.724686;
   DATA[2091,31] := 1.274113;
   DATA[2091,32] := 0.7355248;
   DATA[2091,33] := 0.3065689;
   DATA[2091,34] := 2.0;
   DATA[2091,35] := 250.3845;
   DATA[2091,36] := 1.730048;
   DATA[2091,37] := 189.1182;
   DATA[2091,38] := 0.000128152;
   DATA[2091,39] := 1.0;
   DATA[2091,40] := 1.0;
   DATA[2092,0] := 2.481504;
   DATA[2092,1] := 862.8149;
   DATA[2092,2] := 2.0;
   DATA[2092,3] := 2.0;
   DATA[2092,4] := 262.4007;
   DATA[2092,5] := 8.392271;
   DATA[2092,6] := 330.8639;
   DATA[2092,7] := 2.457694;
   DATA[2092,8] := 2.0;
   DATA[2092,9] := 2.0;
   DATA[2092,10] := 2.0;
   DATA[2092,11] := 19.77079;
   DATA[2092,12] := 2.209909;
   DATA[2092,13] := 805.803;
   DATA[2092,14] := 1.0;
   DATA[2092,15] := 2.0;
   DATA[2092,16] := 1.0;
   DATA[2092,17] := 1.0;
   DATA[2092,18] := 1.0;
   DATA[2092,19] := 2.0;
   DATA[2092,20] := 148.808;
   DATA[2092,21] := 155.0115;
   DATA[2092,22] := 1.718771;
   DATA[2092,23] := 836.4009;
   DATA[2092,24] := 2.0;
   DATA[2092,25] := 2.0;
   DATA[2092,26] := 7.874455;
   DATA[2092,27] := 144.0656;
   DATA[2092,28] := 262.0161;
   DATA[2092,29] := 12.07383;
   DATA[2092,30] := 1.724686;
   DATA[2092,31] := 1.257333;
   DATA[2092,32] := 0.7355248;
   DATA[2092,33] := 0.3065689;
   DATA[2092,34] := 2.0;
   DATA[2092,35] := 250.3845;
   DATA[2092,36] := 1.730048;
   DATA[2092,37] := 189.1182;
   DATA[2092,38] := 0.000128152;
   DATA[2092,39] := 1.0;
   DATA[2092,40] := 1.0;
   DATA[2093,0] := 2.530506;
   DATA[2093,1] := 862.1083;
   DATA[2093,2] := 2.0;
   DATA[2093,3] := 2.0;
   DATA[2093,4] := 262.4007;
   DATA[2093,5] := 8.392271;
   DATA[2093,6] := 330.8639;
   DATA[2093,7] := 2.459616;
   DATA[2093,8] := 2.0;
   DATA[2093,9] := 2.0;
   DATA[2093,10] := 2.0;
   DATA[2093,11] := 19.73238;
   DATA[2093,12] := 2.209909;
   DATA[2093,13] := 806.1635;
   DATA[2093,14] := 1.0;
   DATA[2093,15] := 2.0;
   DATA[2093,16] := 1.0;
   DATA[2093,17] := 1.0;
   DATA[2093,18] := 1.0;
   DATA[2093,19] := 2.0;
   DATA[2093,20] := 148.808;
   DATA[2093,21] := 155.0115;
   DATA[2093,22] := 1.720053;
   DATA[2093,23] := 836.4009;
   DATA[2093,24] := 2.0;
   DATA[2093,25] := 2.0;
   DATA[2093,26] := 7.874455;
   DATA[2093,27] := 144.0656;
   DATA[2093,28] := 262.0161;
   DATA[2093,29] := 12.07383;
   DATA[2093,30] := 1.726737;
   DATA[2093,31] := 1.25349;
   DATA[2093,32] := 0.7355248;
   DATA[2093,33] := 0.3065689;
   DATA[2093,34] := 2.0;
   DATA[2093,35] := 250.3845;
   DATA[2093,36] := 1.730048;
   DATA[2093,37] := 189.1182;
   DATA[2093,38] := 0.000128152;
   DATA[2093,39] := 1.0;
   DATA[2093,40] := 1.0;
   DATA[2094,0] := 2.572783;
   DATA[2094,1] := 862.1083;
   DATA[2094,2] := 2.0;
   DATA[2094,3] := 2.0;
   DATA[2094,4] := 262.4007;
   DATA[2094,5] := 8.392271;
   DATA[2094,6] := 330.8639;
   DATA[2094,7] := 2.460385;
   DATA[2094,8] := 2.0;
   DATA[2094,9] := 2.0;
   DATA[2094,10] := 2.0;
   DATA[2094,11] := 19.73238;
   DATA[2094,12] := 2.209909;
   DATA[2094,13] := 806.0834;
   DATA[2094,14] := 1.0;
   DATA[2094,15] := 2.0;
   DATA[2094,16] := 1.0;
   DATA[2094,17] := 1.0;
   DATA[2094,18] := 1.0;
   DATA[2094,19] := 2.0;
   DATA[2094,20] := 148.808;
   DATA[2094,21] := 155.0115;
   DATA[2094,22] := 1.720053;
   DATA[2094,23] := 836.5932;
   DATA[2094,24] := 2.0;
   DATA[2094,25] := 2.0;
   DATA[2094,26] := 7.874455;
   DATA[2094,27] := 144.0656;
   DATA[2094,28] := 262.0161;
   DATA[2094,29] := 12.07383;
   DATA[2094,30] := 1.728916;
   DATA[2094,31] := 1.260535;
   DATA[2094,32] := 0.7355248;
   DATA[2094,33] := 0.3070813;
   DATA[2094,34] := 2.0;
   DATA[2094,35] := 250.3845;
   DATA[2094,36] := 1.730048;
   DATA[2094,37] := 189.1182;
   DATA[2094,38] := 0.000128152;
   DATA[2094,39] := 1.0;
   DATA[2094,40] := 1.0;
   DATA[2095,0] := 2.606412;
   DATA[2095,1] := 861.9905;
   DATA[2095,2] := 2.0;
   DATA[2095,3] := 2.0;
   DATA[2095,4] := 262.4007;
   DATA[2095,5] := 8.392271;
   DATA[2095,6] := 330.8639;
   DATA[2095,7] := 2.462179;
   DATA[2095,8] := 2.0;
   DATA[2095,9] := 2.0;
   DATA[2095,10] := 2.0;
   DATA[2095,11] := 19.81561;
   DATA[2095,12] := 2.209909;
   DATA[2095,13] := 806.4839;
   DATA[2095,14] := 1.0;
   DATA[2095,15] := 2.0;
   DATA[2095,16] := 1.0;
   DATA[2095,17] := 1.0;
   DATA[2095,18] := 1.0;
   DATA[2095,19] := 2.0;
   DATA[2095,20] := 148.808;
   DATA[2095,21] := 155.0115;
   DATA[2095,22] := 1.720053;
   DATA[2095,23] := 836.2087;
   DATA[2095,24] := 2.0;
   DATA[2095,25] := 2.0;
   DATA[2095,26] := 7.874455;
   DATA[2095,27] := 144.0656;
   DATA[2095,28] := 262.0161;
   DATA[2095,29] := 12.07383;
   DATA[2095,30] := 1.728916;
   DATA[2095,31] := 1.265275;
   DATA[2095,32] := 0.7355248;
   DATA[2095,33] := 0.3070813;
   DATA[2095,34] := 2.0;
   DATA[2095,35] := 250.4646;
   DATA[2095,36] := 1.730048;
   DATA[2095,37] := 189.2784;
   DATA[2095,38] := 0.000128152;
   DATA[2095,39] := 1.0;
   DATA[2095,40] := 1.0;
   DATA[2096,0] := 2.632354;
   DATA[2096,1] := 861.6373;
   DATA[2096,2] := 2.0;
   DATA[2096,3] := 2.0;
   DATA[2096,4] := 262.4007;
   DATA[2096,5] := 8.392271;
   DATA[2096,6] := 330.8639;
   DATA[2096,7] := 2.462179;
   DATA[2096,8] := 2.0;
   DATA[2096,9] := 2.0;
   DATA[2096,10] := 2.0;
   DATA[2096,11] := 19.81561;
   DATA[2096,12] := 2.209909;
   DATA[2096,13] := 806.3638;
   DATA[2096,14] := 1.0;
   DATA[2096,15] := 2.0;
   DATA[2096,16] := 1.0;
   DATA[2096,17] := 1.0;
   DATA[2096,18] := 1.0;
   DATA[2096,19] := 2.0;
   DATA[2096,20] := 148.808;
   DATA[2096,21] := 155.0115;
   DATA[2096,22] := 1.720053;
   DATA[2096,23] := 836.6317;
   DATA[2096,24] := 2.0;
   DATA[2096,25] := 2.0;
   DATA[2096,26] := 7.874455;
   DATA[2096,27] := 144.0656;
   DATA[2096,28] := 262.0161;
   DATA[2096,29] := 12.07383;
   DATA[2096,30] := 1.728916;
   DATA[2096,31] := 1.277443;
   DATA[2096,32] := 0.7355248;
   DATA[2096,33] := 0.3080421;
   DATA[2096,34] := 2.0;
   DATA[2096,35] := 250.5127;
   DATA[2096,36] := 1.730048;
   DATA[2096,37] := 189.2784;
   DATA[2096,38] := 0.000128152;
   DATA[2096,39] := 1.0;
   DATA[2096,40] := 1.0;
   DATA[2097,0] := 2.652532;
   DATA[2097,1] := 861.6373;
   DATA[2097,2] := 2.0;
   DATA[2097,3] := 2.0;
   DATA[2097,4] := 262.4007;
   DATA[2097,5] := 8.392271;
   DATA[2097,6] := 330.8639;
   DATA[2097,7] := 2.462179;
   DATA[2097,8] := 2.0;
   DATA[2097,9] := 2.0;
   DATA[2097,10] := 2.0;
   DATA[2097,11] := 19.81561;
   DATA[2097,12] := 2.209909;
   DATA[2097,13] := 806.4038;
   DATA[2097,14] := 1.0;
   DATA[2097,15] := 2.0;
   DATA[2097,16] := 1.0;
   DATA[2097,17] := 1.0;
   DATA[2097,18] := 1.0;
   DATA[2097,19] := 2.0;
   DATA[2097,20] := 148.808;
   DATA[2097,21] := 155.0115;
   DATA[2097,22] := 1.720053;
   DATA[2097,23] := 836.4394;
   DATA[2097,24] := 2.0;
   DATA[2097,25] := 2.0;
   DATA[2097,26] := 7.874455;
   DATA[2097,27] := 144.0656;
   DATA[2097,28] := 262.0161;
   DATA[2097,29] := 12.07383;
   DATA[2097,30] := 1.728916;
   DATA[2097,31] := 1.287691;
   DATA[2097,32] := 0.7355248;
   DATA[2097,33] := 0.3084265;
   DATA[2097,34] := 2.0;
   DATA[2097,35] := 250.5127;
   DATA[2097,36] := 1.730048;
   DATA[2097,37] := 189.2784;
   DATA[2097,38] := 0.000128152;
   DATA[2097,39] := 1.0;
   DATA[2097,40] := 1.0;
   DATA[2098,0] := 2.658617;
   DATA[2098,1] := 861.127;
   DATA[2098,2] := 2.0;
   DATA[2098,3] := 2.0;
   DATA[2098,4] := 262.4007;
   DATA[2098,5] := 8.392271;
   DATA[2098,6] := 330.8639;
   DATA[2098,7] := 2.462179;
   DATA[2098,8] := 2.0;
   DATA[2098,9] := 2.0;
   DATA[2098,10] := 2.0;
   DATA[2098,11] := 19.81561;
   DATA[2098,12] := 2.209909;
   DATA[2098,13] := 806.564;
   DATA[2098,14] := 1.0;
   DATA[2098,15] := 2.0;
   DATA[2098,16] := 1.0;
   DATA[2098,17] := 1.0;
   DATA[2098,18] := 1.0;
   DATA[2098,19] := 2.0;
   DATA[2098,20] := 148.808;
   DATA[2098,21] := 155.0115;
   DATA[2098,22] := 1.720053;
   DATA[2098,23] := 837.0162;
   DATA[2098,24] := 2.0;
   DATA[2098,25] := 2.0;
   DATA[2098,26] := 7.874455;
   DATA[2098,27] := 144.0913;
   DATA[2098,28] := 262.0161;
   DATA[2098,29] := 12.07383;
   DATA[2098,30] := 1.728916;
   DATA[2098,31] := 1.298962;
   DATA[2098,32] := 0.7355248;
   DATA[2098,33] := 0.3084265;
   DATA[2098,34] := 2.0;
   DATA[2098,35] := 250.3845;
   DATA[2098,36] := 1.730048;
   DATA[2098,37] := 189.2624;
   DATA[2098,38] := 0.000128152;
   DATA[2098,39] := 1.0;
   DATA[2098,40] := 1.0;
   DATA[2099,0] := 2.658617;
   DATA[2099,1] := 861.2448;
   DATA[2099,2] := 2.0;
   DATA[2099,3] := 2.0;
   DATA[2099,4] := 262.4007;
   DATA[2099,5] := 8.392271;
   DATA[2099,6] := 330.8639;
   DATA[2099,7] := 2.462179;
   DATA[2099,8] := 2.0;
   DATA[2099,9] := 2.0;
   DATA[2099,10] := 2.0;
   DATA[2099,11] := 19.81561;
   DATA[2099,12] := 2.209909;
   DATA[2099,13] := 806.8044;
   DATA[2099,14] := 1.0;
   DATA[2099,15] := 2.0;
   DATA[2099,16] := 1.0;
   DATA[2099,17] := 1.0;
   DATA[2099,18] := 1.0;
   DATA[2099,19] := 2.0;
   DATA[2099,20] := 148.808;
   DATA[2099,21] := 155.0115;
   DATA[2099,22] := 1.719284;
   DATA[2099,23] := 836.9393;
   DATA[2099,24] := 2.0;
   DATA[2099,25] := 2.0;
   DATA[2099,26] := 7.874455;
   DATA[2099,27] := 144.0913;
   DATA[2099,28] := 262.0161;
   DATA[2099,29] := 12.07383;
   DATA[2099,30] := 1.728019;
   DATA[2099,31] := 1.301524;
   DATA[2099,32] := 0.7355248;
   DATA[2099,33] := 0.3084265;
   DATA[2099,34] := 2.0;
   DATA[2099,35] := 250.2724;
   DATA[2099,36] := 1.730048;
   DATA[2099,37] := 189.1662;
   DATA[2099,38] := 0.000128152;
   DATA[2099,39] := 1.0;
   DATA[2099,40] := 1.0;
   DATA[2100,0] := 2.630433;
   DATA[2100,1] := 861.0093;
   DATA[2100,2] := 2.0;
   DATA[2100,3] := 2.0;
   DATA[2100,4] := 262.4007;
   DATA[2100,5] := 8.392271;
   DATA[2100,6] := 330.8639;
   DATA[2100,7] := 2.462179;
   DATA[2100,8] := 2.0;
   DATA[2100,9] := 2.0;
   DATA[2100,10] := 2.0;
   DATA[2100,11] := 19.81561;
   DATA[2100,12] := 2.207347;
   DATA[2100,13] := 806.7643;
   DATA[2100,14] := 1.0;
   DATA[2100,15] := 2.0;
   DATA[2100,16] := 1.0;
   DATA[2100,17] := 1.0;
   DATA[2100,18] := 1.0;
   DATA[2100,19] := 2.0;
   DATA[2100,20] := 148.808;
   DATA[2100,21] := 155.0115;
   DATA[2100,22] := 1.717105;
   DATA[2100,23] := 837.17;
   DATA[2100,24] := 2.0;
   DATA[2100,25] := 2.0;
   DATA[2100,26] := 7.874455;
   DATA[2100,27] := 144.0913;
   DATA[2100,28] := 262.0161;
   DATA[2100,29] := 12.07383;
   DATA[2100,30] := 1.724686;
   DATA[2100,31] := 1.302165;
   DATA[2100,32] := 0.7355248;
   DATA[2100,33] := 0.3084265;
   DATA[2100,34] := 2.0;
   DATA[2100,35] := 250.2724;
   DATA[2100,36] := 1.730048;
   DATA[2100,37] := 189.0541;
   DATA[2100,38] := 0.000128152;
   DATA[2100,39] := 1.0;
   DATA[2100,40] := 1.0;
   DATA[2101,0] := 2.623387;
   DATA[2101,1] := 860.8522;
   DATA[2101,2] := 2.0;
   DATA[2101,3] := 2.0;
   DATA[2101,4] := 262.4007;
   DATA[2101,5] := 8.392271;
   DATA[2101,6] := 330.8639;
   DATA[2101,7] := 2.462179;
   DATA[2101,8] := 2.0;
   DATA[2101,9] := 2.0;
   DATA[2101,10] := 2.0;
   DATA[2101,11] := 19.83162;
   DATA[2101,12] := 2.20645;
   DATA[2101,13] := 806.4038;
   DATA[2101,14] := 1.0;
   DATA[2101,15] := 2.0;
   DATA[2101,16] := 1.0;
   DATA[2101,17] := 1.0;
   DATA[2101,18] := 1.0;
   DATA[2101,19] := 2.0;
   DATA[2101,20] := 148.808;
   DATA[2101,21] := 155.0115;
   DATA[2101,22] := 1.717105;
   DATA[2101,23] := 836.9393;
   DATA[2101,24] := 2.0;
   DATA[2101,25] := 2.0;
   DATA[2101,26] := 7.874455;
   DATA[2101,27] := 144.0913;
   DATA[2101,28] := 262.0161;
   DATA[2101,29] := 12.07383;
   DATA[2101,30] := 1.724686;
   DATA[2101,31] := 1.302165;
   DATA[2101,32] := 0.7355248;
   DATA[2101,33] := 0.3084265;
   DATA[2101,34] := 2.0;
   DATA[2101,35] := 250.2724;
   DATA[2101,36] := 1.617916;
   DATA[2101,37] := 189.0541;
   DATA[2101,38] := 0.000128152;
   DATA[2101,39] := 1.0;
   DATA[2101,40] := 1.0;
   DATA[2102,0] := 2.623387;
   DATA[2102,1] := 860.2634;
   DATA[2102,2] := 2.0;
   DATA[2102,3] := 2.0;
   DATA[2102,4] := 262.4007;
   DATA[2102,5] := 8.392271;
   DATA[2102,6] := 330.8639;
   DATA[2102,7] := 2.460641;
   DATA[2102,8] := 2.0;
   DATA[2102,9] := 2.0;
   DATA[2102,10] := 2.0;
   DATA[2102,11] := 19.83162;
   DATA[2102,12] := 2.20645;
   DATA[2102,13] := 806.564;
   DATA[2102,14] := 1.0;
   DATA[2102,15] := 2.0;
   DATA[2102,16] := 1.0;
   DATA[2102,17] := 1.0;
   DATA[2102,18] := 1.0;
   DATA[2102,19] := 2.0;
   DATA[2102,20] := 148.808;
   DATA[2102,21] := 154.7552;
   DATA[2102,22] := 1.717105;
   DATA[2102,23] := 836.8239;
   DATA[2102,24] := 2.0;
   DATA[2102,25] := 2.0;
   DATA[2102,26] := 7.874455;
   DATA[2102,27] := 144.0913;
   DATA[2102,28] := 262.0161;
   DATA[2102,29] := 12.07383;
   DATA[2102,30] := 1.724686;
   DATA[2102,31] := 1.285641;
   DATA[2102,32] := 0.7355248;
   DATA[2102,33] := 0.3084265;
   DATA[2102,34] := 2.0;
   DATA[2102,35] := 250.2724;
   DATA[2102,36] := 1.617916;
   DATA[2102,37] := 189.0541;
   DATA[2102,38] := 0.000128152;
   DATA[2102,39] := 1.0;
   DATA[2102,40] := 1.0;
   DATA[2103,0] := 2.612818;
   DATA[2103,1] := 860.6953;
   DATA[2103,2] := 2.0;
   DATA[2103,3] := 2.0;
   DATA[2103,4] := 262.4007;
   DATA[2103,5] := 8.392271;
   DATA[2103,6] := 330.8639;
   DATA[2103,7] := 2.460641;
   DATA[2103,8] := 2.0;
   DATA[2103,9] := 2.0;
   DATA[2103,10] := 2.0;
   DATA[2103,11] := 19.7996;
   DATA[2103,12] := 2.20645;
   DATA[2103,13] := 806.4038;
   DATA[2103,14] := 1.0;
   DATA[2103,15] := 2.0;
   DATA[2103,16] := 1.0;
   DATA[2103,17] := 1.0;
   DATA[2103,18] := 1.0;
   DATA[2103,19] := 2.0;
   DATA[2103,20] := 148.808;
   DATA[2103,21] := 154.7552;
   DATA[2103,22] := 1.717105;
   DATA[2103,23] := 837.0931;
   DATA[2103,24] := 2.0;
   DATA[2103,25] := 2.0;
   DATA[2103,26] := 7.874455;
   DATA[2103,27] := 144.0913;
   DATA[2103,28] := 262.0161;
   DATA[2103,29] := 12.07383;
   DATA[2103,30] := 1.724686;
   DATA[2103,31] := 1.281158;
   DATA[2103,32] := 0.7355248;
   DATA[2103,33] := 0.3084265;
   DATA[2103,34] := 2.0;
   DATA[2103,35] := 250.2724;
   DATA[2103,36] := 1.617916;
   DATA[2103,37] := 189.0541;
   DATA[2103,38] := 0.000128152;
   DATA[2103,39] := 1.0;
   DATA[2103,40] := 1.0;
   DATA[2104,0] := 2.590398;
   DATA[2104,1] := 860.2634;
   DATA[2104,2] := 2.0;
   DATA[2104,3] := 2.0;
   DATA[2104,4] := 262.4007;
   DATA[2104,5] := 8.392271;
   DATA[2104,6] := 330.8639;
   DATA[2104,7] := 2.460641;
   DATA[2104,8] := 2.0;
   DATA[2104,9] := 2.0;
   DATA[2104,10] := 2.0;
   DATA[2104,11] := 19.7964;
   DATA[2104,12] := 2.20645;
   DATA[2104,13] := 806.524;
   DATA[2104,14] := 1.0;
   DATA[2104,15] := 2.0;
   DATA[2104,16] := 1.0;
   DATA[2104,17] := 1.0;
   DATA[2104,18] := 1.0;
   DATA[2104,19] := 2.0;
   DATA[2104,20] := 148.808;
   DATA[2104,21] := 154.7552;
   DATA[2104,22] := 1.717105;
   DATA[2104,23] := 837.0931;
   DATA[2104,24] := 2.0;
   DATA[2104,25] := 2.0;
   DATA[2104,26] := 7.874455;
   DATA[2104,27] := 144.0913;
   DATA[2104,28] := 262.0161;
   DATA[2104,29] := 12.07383;
   DATA[2104,30] := 1.724686;
   DATA[2104,31] := 1.275394;
   DATA[2104,32] := 0.7355248;
   DATA[2104,33] := 0.3081703;
   DATA[2104,34] := 2.0;
   DATA[2104,35] := 250.2724;
   DATA[2104,36] := 1.617916;
   DATA[2104,37] := 189.0541;
   DATA[2104,38] := 0.000128152;
   DATA[2104,39] := 1.0;
   DATA[2104,40] := 1.0;
   DATA[2105,0] := 2.574064;
   DATA[2105,1] := 860.342;
   DATA[2105,2] := 2.0;
   DATA[2105,3] := 2.0;
   DATA[2105,4] := 262.4007;
   DATA[2105,5] := 8.392271;
   DATA[2105,6] := 330.8639;
   DATA[2105,7] := 2.460641;
   DATA[2105,8] := 2.0;
   DATA[2105,9] := 2.0;
   DATA[2105,10] := 2.0;
   DATA[2105,11] := 19.7964;
   DATA[2105,12] := 2.208244;
   DATA[2105,13] := 806.0834;
   DATA[2105,14] := 1.0;
   DATA[2105,15] := 2.0;
   DATA[2105,16] := 1.0;
   DATA[2105,17] := 1.0;
   DATA[2105,18] := 1.0;
   DATA[2105,19] := 2.0;
   DATA[2105,20] := 148.808;
   DATA[2105,21] := 154.7552;
   DATA[2105,22] := 1.717105;
   DATA[2105,23] := 837.3238;
   DATA[2105,24] := 2.0;
   DATA[2105,25] := 2.0;
   DATA[2105,26] := 7.874455;
   DATA[2105,27] := 144.0913;
   DATA[2105,28] := 262.0161;
   DATA[2105,29] := 12.07383;
   DATA[2105,30] := 1.724686;
   DATA[2105,31] := 1.273601;
   DATA[2105,32] := 0.7355248;
   DATA[2105,33] := 0.3074656;
   DATA[2105,34] := 2.0;
   DATA[2105,35] := 250.2243;
   DATA[2105,36] := 1.617916;
   DATA[2105,37] := 189.0541;
   DATA[2105,38] := 0.000128152;
   DATA[2105,39] := 1.0;
   DATA[2105,40] := 1.0;
   DATA[2106,0] := 2.559331;
   DATA[2106,1] := 860.2634;
   DATA[2106,2] := 2.0;
   DATA[2106,3] := 2.0;
   DATA[2106,4] := 262.4007;
   DATA[2106,5] := 8.392271;
   DATA[2106,6] := 330.8639;
   DATA[2106,7] := 2.460641;
   DATA[2106,8] := 2.0;
   DATA[2106,9] := 2.0;
   DATA[2106,10] := 2.0;
   DATA[2106,11] := 19.7964;
   DATA[2106,12] := 2.209653;
   DATA[2106,13] := 806.3237;
   DATA[2106,14] := 1.0;
   DATA[2106,15] := 2.0;
   DATA[2106,16] := 1.0;
   DATA[2106,17] := 1.0;
   DATA[2106,18] := 1.0;
   DATA[2106,19] := 2.0;
   DATA[2106,20] := 148.808;
   DATA[2106,21] := 154.8065;
   DATA[2106,22] := 1.717105;
   DATA[2106,23] := 837.4007;
   DATA[2106,24] := 2.0;
   DATA[2106,25] := 2.0;
   DATA[2106,26] := 7.874455;
   DATA[2106,27] := 144.0913;
   DATA[2106,28] := 262.0161;
   DATA[2106,29] := 12.07383;
   DATA[2106,30] := 1.724686;
   DATA[2106,31] := 1.277699;
   DATA[2106,32] := 0.7355248;
   DATA[2106,33] := 0.3082983;
   DATA[2106,34] := 2.0;
   DATA[2106,35] := 250.2243;
   DATA[2106,36] := 1.617916;
   DATA[2106,37] := 189.022;
   DATA[2106,38] := 0.000128152;
   DATA[2106,39] := 1.0;
   DATA[2106,40] := 1.0;
   DATA[2107,0] := 2.543958;
   DATA[2107,1] := 860.499;
   DATA[2107,2] := 2.0;
   DATA[2107,3] := 2.0;
   DATA[2107,4] := 262.4007;
   DATA[2107,5] := 8.392271;
   DATA[2107,6] := 330.7357;
   DATA[2107,7] := 2.460641;
   DATA[2107,8] := 2.0;
   DATA[2107,9] := 2.0;
   DATA[2107,10] := 2.0;
   DATA[2107,11] := 19.75479;
   DATA[2107,12] := 2.209653;
   DATA[2107,13] := 806.1635;
   DATA[2107,14] := 1.0;
   DATA[2107,15] := 2.0;
   DATA[2107,16] := 1.0;
   DATA[2107,17] := 1.0;
   DATA[2107,18] := 1.0;
   DATA[2107,19] := 2.0;
   DATA[2107,20] := 148.808;
   DATA[2107,21] := 154.8065;
   DATA[2107,22] := 1.717105;
   DATA[2107,23] := 837.7083;
   DATA[2107,24] := 2.0;
   DATA[2107,25] := 2.0;
   DATA[2107,26] := 7.873174;
   DATA[2107,27] := 144.0913;
   DATA[2107,28] := 262.0161;
   DATA[2107,29] := 12.07383;
   DATA[2107,30] := 1.725583;
   DATA[2107,31] := 1.274241;
   DATA[2107,32] := 0.7355248;
   DATA[2107,33] := 0.3084905;
   DATA[2107,34] := 2.0;
   DATA[2107,35] := 250.2243;
   DATA[2107,36] := 1.617916;
   DATA[2107,37] := 189.022;
   DATA[2107,38] := 0.000128152;
   DATA[2107,39] := 1.0;
   DATA[2107,40] := 1.0;
   DATA[2108,0] := 2.522499;
   DATA[2108,1] := 860.5382;
   DATA[2108,2] := 2.0;
   DATA[2108,3] := 2.0;
   DATA[2108,4] := 262.4007;
   DATA[2108,5] := 8.392271;
   DATA[2108,6] := 330.7357;
   DATA[2108,7] := 2.460641;
   DATA[2108,8] := 2.0;
   DATA[2108,9] := 2.0;
   DATA[2108,10] := 2.0;
   DATA[2108,11] := 19.75479;
   DATA[2108,12] := 2.209653;
   DATA[2108,13] := 806.0834;
   DATA[2108,14] := 1.0;
   DATA[2108,15] := 2.0;
   DATA[2108,16] := 1.0;
   DATA[2108,17] := 1.0;
   DATA[2108,18] := 1.0;
   DATA[2108,19] := 2.0;
   DATA[2108,20] := 148.808;
   DATA[2108,21] := 154.8065;
   DATA[2108,22] := 1.718643;
   DATA[2108,23] := 837.4007;
   DATA[2108,24] := 2.0;
   DATA[2108,25] := 2.0;
   DATA[2108,26] := 7.873174;
   DATA[2108,27] := 144.0913;
   DATA[2108,28] := 262.0161;
   DATA[2108,29] := 12.07383;
   DATA[2108,30] := 1.72725;
   DATA[2108,31] := 1.281542;
   DATA[2108,32] := 0.7355248;
   DATA[2108,33] := 0.3084905;
   DATA[2108,34] := 2.0;
   DATA[2108,35] := 250.2403;
   DATA[2108,36] := 1.617916;
   DATA[2108,37] := 189.022;
   DATA[2108,38] := 0.000128152;
   DATA[2108,39] := 1.0;
   DATA[2108,40] := 1.0;
   DATA[2109,0] := 2.509048;
   DATA[2109,1] := 860.4205;
   DATA[2109,2] := 2.0;
   DATA[2109,3] := 2.0;
   DATA[2109,4] := 262.4007;
   DATA[2109,5] := 8.392271;
   DATA[2109,6] := 330.7357;
   DATA[2109,7] := 2.460641;
   DATA[2109,8] := 2.0;
   DATA[2109,9] := 2.0;
   DATA[2109,10] := 2.0;
   DATA[2109,11] := 19.75479;
   DATA[2109,12] := 2.209525;
   DATA[2109,13] := 805.9232;
   DATA[2109,14] := 1.0;
   DATA[2109,15] := 2.0;
   DATA[2109,16] := 1.0;
   DATA[2109,17] := 1.0;
   DATA[2109,18] := 1.0;
   DATA[2109,19] := 2.0;
   DATA[2109,20] := 148.808;
   DATA[2109,21] := 154.8065;
   DATA[2109,22] := 1.718643;
   DATA[2109,23] := 837.516;
   DATA[2109,24] := 2.0;
   DATA[2109,25] := 2.0;
   DATA[2109,26] := 7.873174;
   DATA[2109,27] := 144.0913;
   DATA[2109,28] := 262.0161;
   DATA[2109,29] := 12.07383;
   DATA[2109,30] := 1.727378;
   DATA[2109,31] := 1.281542;
   DATA[2109,32] := 0.7355248;
   DATA[2109,33] := 0.3084905;
   DATA[2109,34] := 2.0;
   DATA[2109,35] := 250.3204;
   DATA[2109,36] := 1.69801;
   DATA[2109,37] := 189.022;
   DATA[2109,38] := 0.000128152;
   DATA[2109,39] := 1.0;
   DATA[2109,40] := 1.0;
   DATA[2110,0] := 2.493034;
   DATA[2110,1] := 860.813;
   DATA[2110,2] := 2.0;
   DATA[2110,3] := 2.0;
   DATA[2110,4] := 262.4007;
   DATA[2110,5] := 8.392271;
   DATA[2110,6] := 330.7357;
   DATA[2110,7] := 2.460641;
   DATA[2110,8] := 2.0;
   DATA[2110,9] := 2.0;
   DATA[2110,10] := 2.0;
   DATA[2110,11] := 19.75479;
   DATA[2110,12] := 2.207091;
   DATA[2110,13] := 805.5627;
   DATA[2110,14] := 1.0;
   DATA[2110,15] := 2.0;
   DATA[2110,16] := 1.0;
   DATA[2110,17] := 1.0;
   DATA[2110,18] := 1.0;
   DATA[2110,19] := 2.0;
   DATA[2110,20] := 148.808;
   DATA[2110,21] := 154.8065;
   DATA[2110,22] := 1.718643;
   DATA[2110,23] := 837.4007;
   DATA[2110,24] := 2.0;
   DATA[2110,25] := 2.0;
   DATA[2110,26] := 7.873174;
   DATA[2110,27] := 144.0913;
   DATA[2110,28] := 262.0161;
   DATA[2110,29] := 12.07383;
   DATA[2110,30] := 1.727378;
   DATA[2110,31] := 1.264634;
   DATA[2110,32] := 0.7355248;
   DATA[2110,33] := 0.3084905;
   DATA[2110,34] := 2.0;
   DATA[2110,35] := 250.4005;
   DATA[2110,36] := 1.746067;
   DATA[2110,37] := 189.1983;
   DATA[2110,38] := 0.000128152;
   DATA[2110,39] := 1.0;
   DATA[2110,40] := 1.0;
   DATA[2111,0] := 2.4767;
   DATA[2111,1] := 860.8915;
   DATA[2111,2] := 2.0;
   DATA[2111,3] := 2.0;
   DATA[2111,4] := 262.4007;
   DATA[2111,5] := 8.392271;
   DATA[2111,6] := 330.7357;
   DATA[2111,7] := 2.460641;
   DATA[2111,8] := 2.0;
   DATA[2111,9] := 2.0;
   DATA[2111,10] := 2.0;
   DATA[2111,11] := 19.68436;
   DATA[2111,12] := 2.207091;
   DATA[2111,13] := 805.8831;
   DATA[2111,14] := 1.0;
   DATA[2111,15] := 2.0;
   DATA[2111,16] := 1.0;
   DATA[2111,17] := 1.0;
   DATA[2111,18] := 1.0;
   DATA[2111,19] := 2.0;
   DATA[2111,20] := 148.808;
   DATA[2111,21] := 154.8065;
   DATA[2111,22] := 1.718643;
   DATA[2111,23] := 837.5544;
   DATA[2111,24] := 2.0;
   DATA[2111,25] := 2.0;
   DATA[2111,26] := 7.873174;
   DATA[2111,27] := 144.0913;
   DATA[2111,28] := 262.0161;
   DATA[2111,29] := 12.07383;
   DATA[2111,30] := 1.727378;
   DATA[2111,31] := 1.261048;
   DATA[2111,32] := 0.7353967;
   DATA[2111,33] := 0.3084905;
   DATA[2111,34] := 2.0;
   DATA[2111,35] := 250.4005;
   DATA[2111,36] := 1.746067;
   DATA[2111,37] := 189.1983;
   DATA[2111,38] := 0.000128152;
   DATA[2111,39] := 1.0;
   DATA[2111,40] := 1.0;
   DATA[2112,0] := 2.4767;
   DATA[2112,1] := 860.8915;
   DATA[2112,2] := 2.0;
   DATA[2112,3] := 2.0;
   DATA[2112,4] := 262.4007;
   DATA[2112,5] := 8.392271;
   DATA[2112,6] := 330.7357;
   DATA[2112,7] := 2.460641;
   DATA[2112,8] := 2.0;
   DATA[2112,9] := 2.0;
   DATA[2112,10] := 2.0;
   DATA[2112,11] := 19.68436;
   DATA[2112,12] := 2.207091;
   DATA[2112,13] := 805.8831;
   DATA[2112,14] := 1.0;
   DATA[2112,15] := 2.0;
   DATA[2112,16] := 1.0;
   DATA[2112,17] := 1.0;
   DATA[2112,18] := 1.0;
   DATA[2112,19] := 2.0;
   DATA[2112,20] := 148.808;
   DATA[2112,21] := 154.8065;
   DATA[2112,22] := 1.718643;
   DATA[2112,23] := 837.5544;
   DATA[2112,24] := 2.0;
   DATA[2112,25] := 2.0;
   DATA[2112,26] := 7.873174;
   DATA[2112,27] := 144.0913;
   DATA[2112,28] := 262.0161;
   DATA[2112,29] := 12.07383;
   DATA[2112,30] := 1.727378;
   DATA[2112,31] := 1.261048;
   DATA[2112,32] := 0.7353967;
   DATA[2112,33] := 0.3084905;
   DATA[2112,34] := 2.0;
   DATA[2112,35] := 250.4005;
   DATA[2112,36] := 1.746067;
   DATA[2112,37] := 189.1983;
   DATA[2112,38] := 0.000128152;
   DATA[2112,39] := 1.0;
   DATA[2112,40] := 1.0;
   DATA[2113,0] := 2.455882;
   DATA[2113,1] := 861.127;
   DATA[2113,2] := 2.0;
   DATA[2113,3] := 2.0;
   DATA[2113,4] := 262.4007;
   DATA[2113,5] := 8.392271;
   DATA[2113,6] := 330.7357;
   DATA[2113,7] := 2.460641;
   DATA[2113,8] := 2.0;
   DATA[2113,9] := 2.0;
   DATA[2113,10] := 2.0;
   DATA[2113,11] := 19.68436;
   DATA[2113,12] := 2.207091;
   DATA[2113,13] := 805.6829;
   DATA[2113,14] := 1.0;
   DATA[2113,15] := 2.0;
   DATA[2113,16] := 1.0;
   DATA[2113,17] := 1.0;
   DATA[2113,18] := 1.0;
   DATA[2113,19] := 2.0;
   DATA[2113,20] := 148.808;
   DATA[2113,21] := 154.8065;
   DATA[2113,22] := 1.717489;
   DATA[2113,23] := 837.2853;
   DATA[2113,24] := 2.0;
   DATA[2113,25] := 2.0;
   DATA[2113,26] := 7.873174;
   DATA[2113,27] := 144.0913;
   DATA[2113,28] := 262.0161;
   DATA[2113,29] := 12.07383;
   DATA[2113,30] := 1.727378;
   DATA[2113,31] := 1.255924;
   DATA[2113,32] := 0.7353967;
   DATA[2113,33] := 0.306761;
   DATA[2113,34] := 2.0;
   DATA[2113,35] := 250.4005;
   DATA[2113,36] := 1.746067;
   DATA[2113,37] := 189.1983;
   DATA[2113,38] := 0.000128152;
   DATA[2113,39] := 1.0;
   DATA[2113,40] := 1.0;
   DATA[2114,0] := 2.443391;
   DATA[2114,1] := 861.0878;
   DATA[2114,2] := 2.0;
   DATA[2114,3] := 2.0;
   DATA[2114,4] := 262.4007;
   DATA[2114,5] := 8.392271;
   DATA[2114,6] := 330.7357;
   DATA[2114,7] := 2.460641;
   DATA[2114,8] := 2.0;
   DATA[2114,9] := 2.0;
   DATA[2114,10] := 2.0;
   DATA[2114,11] := 19.68436;
   DATA[2114,12] := 2.207731;
   DATA[2114,13] := 805.7229;
   DATA[2114,14] := 1.0;
   DATA[2114,15] := 2.0;
   DATA[2114,16] := 1.0;
   DATA[2114,17] := 1.0;
   DATA[2114,18] := 1.0;
   DATA[2114,19] := 2.0;
   DATA[2114,20] := 148.808;
   DATA[2114,21] := 154.8065;
   DATA[2114,22] := 1.717489;
   DATA[2114,23] := 837.7083;
   DATA[2114,24] := 2.0;
   DATA[2114,25] := 2.0;
   DATA[2114,26] := 7.873174;
   DATA[2114,27] := 144.0913;
   DATA[2114,28] := 262.0161;
   DATA[2114,29] := 12.07383;
   DATA[2114,30] := 1.727378;
   DATA[2114,31] := 1.255156;
   DATA[2114,32] := 0.7353967;
   DATA[2114,33] := 0.306761;
   DATA[2114,34] := 2.0;
   DATA[2114,35] := 250.4005;
   DATA[2114,36] := 1.746067;
   DATA[2114,37] := 189.1983;
   DATA[2114,38] := 0.000128152;
   DATA[2114,39] := 1.0;
   DATA[2114,40] := 1.0;
   DATA[2115,0] := 2.42994;
   DATA[2115,1] := 861.2055;
   DATA[2115,2] := 2.0;
   DATA[2115,3] := 2.0;
   DATA[2115,4] := 262.4007;
   DATA[2115,5] := 8.392271;
   DATA[2115,6] := 330.7357;
   DATA[2115,7] := 2.460641;
   DATA[2115,8] := 2.0;
   DATA[2115,9] := 2.0;
   DATA[2115,10] := 2.0;
   DATA[2115,11] := 19.68436;
   DATA[2115,12] := 2.209013;
   DATA[2115,13] := 805.4826;
   DATA[2115,14] := 1.0;
   DATA[2115,15] := 2.0;
   DATA[2115,16] := 1.0;
   DATA[2115,17] := 1.0;
   DATA[2115,18] := 1.0;
   DATA[2115,19] := 2.0;
   DATA[2115,20] := 148.808;
   DATA[2115,21] := 154.8065;
   DATA[2115,22] := 1.717489;
   DATA[2115,23] := 837.6698;
   DATA[2115,24] := 2.0;
   DATA[2115,25] := 2.0;
   DATA[2115,26] := 7.873174;
   DATA[2115,27] := 144.0913;
   DATA[2115,28] := 262.0161;
   DATA[2115,29] := 12.07383;
   DATA[2115,30] := 1.727378;
   DATA[2115,31] := 1.274625;
   DATA[2115,32] := 0.7353967;
   DATA[2115,33] := 0.306761;
   DATA[2115,34] := 2.0;
   DATA[2115,35] := 250.4005;
   DATA[2115,36] := 1.746067;
   DATA[2115,37] := 189.1182;
   DATA[2115,38] := 0.000128152;
   DATA[2115,39] := 1.0;
   DATA[2115,40] := 1.0;
   DATA[2116,0] := 2.423854;
   DATA[2116,1] := 861.2448;
   DATA[2116,2] := 2.0;
   DATA[2116,3] := 2.0;
   DATA[2116,4] := 262.4007;
   DATA[2116,5] := 8.392271;
   DATA[2116,6] := 330.7357;
   DATA[2116,7] := 2.460641;
   DATA[2116,8] := 2.0;
   DATA[2116,9] := 2.0;
   DATA[2116,10] := 2.0;
   DATA[2116,11] := 19.68436;
   DATA[2116,12] := 2.209013;
   DATA[2116,13] := 805.7229;
   DATA[2116,14] := 1.0;
   DATA[2116,15] := 2.0;
   DATA[2116,16] := 1.0;
   DATA[2116,17] := 1.0;
   DATA[2116,18] := 1.0;
   DATA[2116,19] := 2.0;
   DATA[2116,20] := 148.808;
   DATA[2116,21] := 154.8065;
   DATA[2116,22] := 1.717489;
   DATA[2116,23] := 837.9774;
   DATA[2116,24] := 2.0;
   DATA[2116,25] := 2.0;
   DATA[2116,26] := 7.873174;
   DATA[2116,27] := 144.2451;
   DATA[2116,28] := 262.0161;
   DATA[2116,29] := 12.07383;
   DATA[2116,30] := 1.727378;
   DATA[2116,31] := 1.283079;
   DATA[2116,32] := 0.7353967;
   DATA[2116,33] := 0.306761;
   DATA[2116,34] := 2.0;
   DATA[2116,35] := 250.4005;
   DATA[2116,36] := 1.746067;
   DATA[2116,37] := 189.1182;
   DATA[2116,38] := 0.000128152;
   DATA[2116,39] := 1.0;
   DATA[2116,40] := 1.0;
   DATA[2117,0] := 2.423854;
   DATA[2117,1] := 861.6765;
   DATA[2117,2] := 2.0;
   DATA[2117,3] := 2.0;
   DATA[2117,4] := 262.4007;
   DATA[2117,5] := 8.392271;
   DATA[2117,6] := 330.7357;
   DATA[2117,7] := 2.463204;
   DATA[2117,8] := 2.0;
   DATA[2117,9] := 2.0;
   DATA[2117,10] := 2.0;
   DATA[2117,11] := 19.68436;
   DATA[2117,12] := 2.209013;
   DATA[2117,13] := 805.6829;
   DATA[2117,14] := 1.0;
   DATA[2117,15] := 2.0;
   DATA[2117,16] := 1.0;
   DATA[2117,17] := 1.0;
   DATA[2117,18] := 1.0;
   DATA[2117,19] := 2.0;
   DATA[2117,20] := 148.808;
   DATA[2117,21] := 154.8065;
   DATA[2117,22] := 1.717489;
   DATA[2117,23] := 837.9774;
   DATA[2117,24] := 2.0;
   DATA[2117,25] := 2.0;
   DATA[2117,26] := 7.873174;
   DATA[2117,27] := 144.322;
   DATA[2117,28] := 262.0161;
   DATA[2117,29] := 12.03538;
   DATA[2117,30] := 1.727378;
   DATA[2117,31] := 1.290124;
   DATA[2117,32] := 0.7353967;
   DATA[2117,33] := 0.306761;
   DATA[2117,34] := 2.0;
   DATA[2117,35] := 250.4005;
   DATA[2117,36] := 1.746067;
   DATA[2117,37] := 189.1182;
   DATA[2117,38] := 0.000128152;
   DATA[2117,39] := 1.0;
   DATA[2117,40] := 1.0;
   DATA[2118,0] := 2.448836;
   DATA[2118,1] := 861.2448;
   DATA[2118,2] := 2.0;
   DATA[2118,3] := 2.0;
   DATA[2118,4] := 262.4007;
   DATA[2118,5] := 8.392271;
   DATA[2118,6] := 330.7357;
   DATA[2118,7] := 2.463204;
   DATA[2118,8] := 2.0;
   DATA[2118,9] := 2.0;
   DATA[2118,10] := 2.0;
   DATA[2118,11] := 19.68436;
   DATA[2118,12] := 2.209013;
   DATA[2118,13] := 805.7229;
   DATA[2118,14] := 1.0;
   DATA[2118,15] := 2.0;
   DATA[2118,16] := 1.0;
   DATA[2118,17] := 1.0;
   DATA[2118,18] := 1.0;
   DATA[2118,19] := 2.0;
   DATA[2118,20] := 148.808;
   DATA[2118,21] := 154.8065;
   DATA[2118,22] := 1.717489;
   DATA[2118,23] := 838.4773;
   DATA[2118,24] := 2.0;
   DATA[2118,25] := 2.0;
   DATA[2118,26] := 7.873174;
   DATA[2118,27] := 144.322;
   DATA[2118,28] := 262.0161;
   DATA[2118,29] := 12.03538;
   DATA[2118,30] := 1.727378;
   DATA[2118,31] := 1.291789;
   DATA[2118,32] := 0.7353967;
   DATA[2118,33] := 0.306761;
   DATA[2118,34] := 2.0;
   DATA[2118,35] := 250.1122;
   DATA[2118,36] := 1.746067;
   DATA[2118,37] := 189.0381;
   DATA[2118,38] := 0.000128152;
   DATA[2118,39] := 1.0;
   DATA[2118,40] := 1.0;
   DATA[2119,0] := 2.493034;
   DATA[2119,1] := 861.7943;
   DATA[2119,2] := 2.0;
   DATA[2119,3] := 2.0;
   DATA[2119,4] := 262.4007;
   DATA[2119,5] := 8.392271;
   DATA[2119,6] := 330.7357;
   DATA[2119,7] := 2.463204;
   DATA[2119,8] := 2.0;
   DATA[2119,9] := 2.0;
   DATA[2119,10] := 2.0;
   DATA[2119,11] := 19.68436;
   DATA[2119,12] := 2.209013;
   DATA[2119,13] := 806.0033;
   DATA[2119,14] := 1.0;
   DATA[2119,15] := 2.0;
   DATA[2119,16] := 1.0;
   DATA[2119,17] := 1.0;
   DATA[2119,18] := 1.0;
   DATA[2119,19] := 2.0;
   DATA[2119,20] := 148.808;
   DATA[2119,21] := 154.8065;
   DATA[2119,22] := 1.717489;
   DATA[2119,23] := 838.285;
   DATA[2119,24] := 2.0;
   DATA[2119,25] := 2.0;
   DATA[2119,26] := 7.873174;
   DATA[2119,27] := 144.322;
   DATA[2119,28] := 262.0161;
   DATA[2119,29] := 12.03538;
   DATA[2119,30] := 1.72725;
   DATA[2119,31] := 1.288075;
   DATA[2119,32] := 0.7353967;
   DATA[2119,33] := 0.306761;
   DATA[2119,34] := 2.0;
   DATA[2119,35] := 250.1122;
   DATA[2119,36] := 1.69801;
   DATA[2119,37] := 189.0381;
   DATA[2119,38] := 0.000128152;
   DATA[2119,39] := 1.0;
   DATA[2119,40] := 1.0;
   DATA[2120,0] := 2.536271;
   DATA[2120,1] := 862.2653;
   DATA[2120,2] := 2.0;
   DATA[2120,3] := 2.0;
   DATA[2120,4] := 262.4007;
   DATA[2120,5] := 8.392271;
   DATA[2120,6] := 330.7357;
   DATA[2120,7] := 2.461923;
   DATA[2120,8] := 2.0;
   DATA[2120,9] := 2.0;
   DATA[2120,10] := 2.0;
   DATA[2120,11] := 19.72598;
   DATA[2120,12] := 2.209013;
